*)
(* berechne den 1.1 des jahres von idate. *)
yr := year(idate);
d1 := year_begin(yr);
(* wochentag von d1 *)
w1 := weekday(d1);
(* offset des montags der eletzten KW des vorjahres *)
(* wenn der erste tag des jahres größer als donnerstag ist dann beginnt die letzte kw am montag davor *)
(* wenn der erste tag des jahres ein donnerstag oder kleiner ist beginnt die erste kw 2 montage davor *)
IF w1 < 5 THEN
	ds := DATE_TO_DWORD(d1) - (w1+6) * 86400;
ELSE
	ds := DATE_TO_DWORD(d1) + (1-w1) * 86400;
END_IF;

(* kalenderwoche des eingangsdatums *)
work_week := DWORD_TO_INT((DATE_TO_DWORD(idate) - ds) / 604800);

(* korrektur wenn work_week = 0 *)
IF work_week = 0 THEN
	(* work_week needs to be 53 when 1.jan of the year before is thursday or dec 31. is thursday. *)
	(* first and last weekday of a year is equal and one more day for a leap_year. *)
	IF w1 > 1 THEN w31 := w1 - 1; ELSE W31 := 7; END_IF;
	IF leap_year(yr - 1) THEN IF w31 > 1 THEN w01 := W31 - 1; ELSE w1 := 7; END_IF; END_IF;
	(* if first or last day of a year is a thursday, the year has 53 weeks *)
	IF w31 = 4 OR w01 = 4 THEN work_week := 53; ELSE work_week := 52; END_IF;
ELSE
	(* end of year calculation *)
	(* calculated the first and last weekday *)
	IF leap_year(yr) THEN
		IF w1 < 7 THEN w31 := w1 + 1; ELSE w31 := 1; END_IF;
	ELSE
		w31 := w1;
	END_IF;
	(* if first or last day is thursday then the year has 53 weeks otherwise only 52 *)
	IF w31 = 4 OR w1 = 4 THEN wm := 53; ELSE wm := 52; END_IF;
	IF work_week > wm THEN work_week := 1; END_IF;
END_IF;



(* old code before rev 1.2
w1 := weekday(set_Date(year(idate), 1,1));
IF w1 < 5 THEN
	work_week := (day_of_year(idate) + w1 + 5)/7;
ELSE
	work_week := (day_of_year(idate) + w1 - 2)/7;
END_IF
*)


(* revision history

hm 17.1.2007		rev 1.1
	deleted unused variable yday

hm	19. dec 2007	rev 1.2
	changed code for better performance
	changed code to comply with ISO8601
*)
END_FUNCTION

(* POU String/FIND_CHAR, ST *)
FUNCTION FIND_CHAR : INT
VAR_INPUT
	str : STRING;
	pos : INT;
END_VAR
VAR
	i: INT;
	pt : POINTER TO ARRAY[1..255] OF BYTE;
	stop: INT;
	X: BYTE;
END_VAR

(*
version 1.0	29. feb 2008
programmer 	hugo
tested by		tobias

find_char searches str and returns the starting position of the first character that is not a control character.
control characters are the ascii character 00 .. 31.

*)
pt := ADR(str);
stop := LEN(str);
FOR i := MAX(pos,1) TO stop DO;
	X := pt^[i];
	IF X > 31 THEN
		FIND_CHAR := i;
		RETURN;
	END_IF;
END_FOR;
FIND_CHAR := 0;


(* revision history
hm		29. feb 2008	rev 1.0
	original version

*)
END_FUNCTION

(* POU String/FIND_CTRL, ST *)
FUNCTION FIND_CTRL : INT
VAR_INPUT
	str : STRING;
	pos : INT;
END_VAR
VAR
	i: INT;
	pt : POINTER TO ARRAY[1..255] OF BYTE;
	stop: INT;
	x: BYTE;
END_VAR

(*
version 1.0	29. feb 2008
programmer 	hugo
tested by		tobias

find_ctrl searches str and returns the starting position of a control character
control characters are the ascii character 00 .. 31.

*)
pt := ADR(str);
stop := LEN(str);
FOR i := MAX(pos,1) TO stop DO;
	x := PT^[I];
	IF x < 32 THEN
		FIND_CTRL := i;
		RETURN;
	END_IF;
END_FOR;
FIND_CTRL := 0;


(* revision history
hm		29. feb 2008	rev 1.0
	original version

*)
END_FUNCTION

(* POU String/FINDP, ST *)
FUNCTION FINDP : INT
VAR_INPUT
	str : STRING;
	src : STRING;
	pos: INT;
END_VAR
VAR
	i: INT;
	ls: INT;
	lx: INT;
	stp: INT;
END_VAR

(*
version 1.1	29. feb 2009
programmer 	hugo
tested by		tobias

the function findP searches a string str for the occurence of src beginning at the position pos.

*)
ls := LEN(str);
lx := LEN(src);
IF ls < lx OR lx = 0 THEN RETURN; END_IF;
stp := ls - lx + 1;
FOR i := MAX(pos,1) TO stp DO
	IF MID(str,lx,i) = src THEN
		FINDP := i;
		RETURN;
	END_IF;
END_FOR;
FINDP := 0;

(* revision histroy
hm		4. feb. 2008	rev 1.0
	original release

hm		29. feb 2008	rev 1.1
	ADDED MAX(pos,1) in loop initialization

*)	
END_FUNCTION

(* POU XTEST/Ideas/FM_INVSQRT, ST *)
FUNCTION FM_INVSQRT : REAL
VAR_INPUT
	X: REAL;
END_VAR
VAR
	PTR : POINTER TO DWORD;
	XHALF: REAL;
END_VAR
XHALF := X * 0.5;
ptr := ADR(X);
ptr^ := 16#5F375A86 - SHR(ptr^,1);
FM_INVSQRT := X * (1.5 - XHALF * X * X);
END_FUNCTION

(* POU XTEST/Ideas/I2C, ST *)
FUNCTION_BLOCK I2C
VAR_INPUT
	scl_in : BOOL;
	sda_in : BOOL;
END_VAR
VAR_OUTPUT
	scl_out : BOOL;
	sda_out : BOOL;
	busy: BOOL;
	error: BOOL;
END_VAR
VAR
	state : INT;
END_VAR
(* the following state machine is responsible for all actions on the I2C Bus *)
CASE state OF
	0:	(* no actions *)
		busy := FALSE;

	1: (* ready for transfer *)
		RETURN;

	10: (* generate start condition *)
		busy := TRUE;
		IF sda_in AND scl_in THEN
			(* bus is free, start sequence can be completed *)
			sda_out := FALSE;
			state := 11;
		ELSIF NOT scl_in AND sda_in THEN
			(* if scl is low and sda is true then scl needs to go high first *)
			scl_out := TRUE;
		ELSIF NOT scl_in AND NOT sda_in THEN
			(* both scl and sda are low sda need to go high first *)
			sda_out := TRUE;
		ELSIF NOT scl_in AND NOT sda_in THEN
			(* both scl and sda are low scl need to go low first *)
			scl_out := FALSE;
		END_IF;
	11: (* second phase of start cycle, pull scl low *)
		scl_out := FALSE;
		state := 1;

	20:	(* generate stop condition *)
		busy := TRUE;
		IF scl_in AND NOT sda_in THEN
			(* scl is high and sda is low sequence can be completed *)
			sda_out := TRUE;
			state := 0;
		ELSIF NOT scl_in AND NOT sda_in THEN
			(* scl and sda are low,  scl need to go high first *)
			scl_out := TRUE;
		ELSIF NOT scl_in AND sda_in THEN
			(* scl is low and sda is high, sda need to go low first *)
			sda_out := FALSE;
		ELSIF scl_in AND sda_in THEN
			(* scl and sda are high, scl need to go low first *)
			scl_out := FALSE;
		END_IF;

	30:	(* master acknowledge cycle *)
		IF NOT busy AND scl_in THEN
			(* if no transfer takes place an acknowledge cannot be received *)
			error := TRUE;
		ELSIF TRUE THEN
			(* bring sda true to check for ack *)
			sda_out := TRUE;
		END_IF;



END_CASE
END_FUNCTION_BLOCK

(* POU Network/IP4_CHECK, ST *)
FUNCTION IP4_CHECK : BOOL
VAR_INPUT
	NIP : DWORD;
	LIP : DWORD;
	SM : DWORD;
END_VAR
VAR
END_VAR

(*
version 1.0	4. mar 2008
programmer 	hugo
tested by		oscat

IP4_CHECK testet ob eine Network IP und Local_IP im selben Subnet sind.

*)
IP4_CHECK := (NIP AND sm) = (LIP AND SM);


(* revision history
hm		4. mar 2008	rev 1.0
	original version

*)
END_FUNCTION

(* POU Network/IP4_DECODE, ST *)
FUNCTION IP4_DECODE : DWORD
VAR_INPUT
	str : STRING;
END_VAR
VAR
	d1, d2, d3, d4 : INT;
	s1, s2, s3, s4 : STRING(3);
END_VAR

(*
version 1.0	29. feb 2008
programmer 		kurt
tested by		hugo

IP4_DECODE testet ob ein string eine gültige IPv4 Adresse enthält und gibt die 4 Bytes der IP Adresse als DWORD zurück.

*)
IP4_DECODE := 0;
(* check wheather 3 dots are present *)
IF COUNT_CHAR(str,46) <> 3 THEN RETURN; END_IF;
(* store the positions of the 3 dots *)
d1 := FINDP(str,'.',1);
d2 := FINDP(str,'.',d1+1);
d3 := FINDP(str,'.',d2+1);
IF d1 > 4 OR d2 - d1 > 4 OR d3 - d2 > 4 THEN RETURN; END_IF;
(* store the 3 strings between the dots in d1 .. d4 *)
s1 := LEFT(str,d1-1);
s2 := MID(str,d2-d1-1,d1+1);
s3 := MID(str,d3-d2-1,d2+1);
s4 := RIGHT(str,LEN(str)-d3);
(* check if the 3 strings are numbers only *)
IF NOT IS_NUM(s1) OR NOT IS_NUM(s2) OR NOT IS_NUM(s3) OR NOT IS_NUM(s4) THEN RETURN; END_IF;
(* convert the 4 numbers and check range 0..255 *)
d1 := STRING_TO_INT(s1);
d2 := STRING_TO_INT(s2);
d3 := STRING_TO_INT(s3);
d4 := STRING_TO_INT(s4);
(* check range of numbers *)
IF d1 > 255 OR d2 > 255 OR d3 > 255 OR d4 > 255 THEN RETURN; END_IF;
(* convert to output *)
IP4_DECODE := SHL(INT_TO_DWORD(d1),24) OR SHL(INT_TO_DWORD(d2),16) OR SHL(INT_TO_DWORD(d3),8) OR INT_TO_DWORD(d4);



(* revision history
hm		29. feb 2008	rev 1.0
	original version

*)
END_FUNCTION

(* POU String/IS_NUM, ST *)
FUNCTION IS_NUM : BOOL
VAR_INPUT
	str : STRING;
END_VAR
VAR
	L : INT;
	pt : POINTER TO BYTE;
	pos: INT;
END_VAR

(*
version 1.0	29. feb 2008
programmer 		kurt
tested by		hugo

IS_NUM testet ob in einem string nur Zahlen 0..9 vorkommen.

*)
PT := ADR(str);
L := LEN(str);
FOR pos := 1 TO L DO
	IF NOT (ISC_NUM(pt^)) THEN
		IS_NUM := FALSE;
		RETURN;
	END_IF;
    	PT := PT + 1;
END_FOR;
IS_NUM := L > 0;


(* revision history
hm		29. feb 2008	rev 1.0
	original version

*)
END_FUNCTION

(* POU String/ISC_NUM, ST *)
FUNCTION ISC_NUM : BOOL
VAR_INPUT
	IN : BYTE;
END_VAR
VAR
END_VAR

(*
version 1.0	6. mar 2008
programmer 	oscat
tested by		hugo

ISC_NUM checks if a character is 0..9.

*)
ISC_NUM := IN > 47 AND IN < 58;

(* revision history
hm		6. mar. 2008	rev 1.0
	original version

*)
END_FUNCTION

(* POU Device Drivers/IRTRANS_1, ST *)
FUNCTION_BLOCK IRTRANS_1
VAR_INPUT CONSTANT
	device_code : STRING;
	key_code : STRING;
END_VAR
VAR_INPUT
	cmd : BOOL;
END_VAR
VAR_IN_OUT
	device : STRING;
	key : STRING;
END_VAR
VAR_OUTPUT
	Q : BOOL;
END_VAR
VAR
END_VAR

(*
	version 1.0	2 jan 2008
	programmer 	hugo
	tested BY		tobias

*)
IF cmd AND device_code = device AND key_code = key THEN
	Q := TRUE;
ELSE
	Q := FALSE;
END_IF;

(* revision history
hm	2. jan 2008		rev 1.0
	original version

*)
END_FUNCTION_BLOCK

(* POU Device Drivers/IRTRANS_4, ST *)
FUNCTION_BLOCK IRTRANS_4
VAR_INPUT CONSTANT
	device_code : STRING;
	key_code_0 : STRING;
	key_code_1 : STRING;
	key_code_2 : STRING;
	key_code_3 : STRING;
END_VAR
VAR_INPUT
	cmd : BOOL;
END_VAR
VAR_IN_OUT
	device : STRING;
	key : STRING;
END_VAR
VAR_OUTPUT
	Q0, Q1, Q2, Q3 : BOOL;
END_VAR
VAR
END_VAR

(*
	version 1.0	2 jan 2008
	programmer 	hugo
	tested BY		tobias

*)
Q0 := FALSE;
Q1 := FALSE;
Q2 := FALSE;
Q3 := FALSE;
IF cmd AND device_code = device THEN
	IF key = key_code_0 THEN q0 := TRUE;
	ELSIF key = key_code_1 THEN q1 := TRUE;
	ELSIF key = key_code_2 THEN q2 := TRUE;
	ELSIF key = key_code_3 THEN q3 := TRUE;
	END_IF;
END_IF;

(* revision history
hm	2. jan 2008		rev 1.0
	original version

*)
END_FUNCTION_BLOCK

(* POU Device Drivers/IRTRANS_8, ST *)
FUNCTION_BLOCK IRTRANS_8
VAR_INPUT CONSTANT
	device_code : STRING;
	key_code_0 : STRING;
	key_code_1 : STRING;
	key_code_2 : STRING;
	key_code_3 : STRING;
	key_code_4 : STRING;
	key_code_5 : STRING;
	key_code_6 : STRING;
	key_code_7 : STRING;
END_VAR
VAR_INPUT
	cmd : BOOL;
END_VAR
VAR_IN_OUT
	device : STRING;
	key : STRING;
END_VAR
VAR_OUTPUT
	Q0, Q1, Q2, Q3, Q4, Q5, Q6, Q7 : BOOL;
END_VAR
VAR
END_VAR

(*
	version 1.0	2 jan 2008
	programmer 	hugo
	tested BY		tobias

*)
Q0 := FALSE;
Q1 := FALSE;
Q2 := FALSE;
Q3 := FALSE;
Q4 := FALSE;
Q5 := FALSE;
Q6 := FALSE;
Q7 := FALSE;
IF cmd AND device_code = device THEN
	IF key = key_code_0 THEN q0 := TRUE;
	ELSIF key = key_code_1 THEN q1 := TRUE;
	ELSIF key = key_code_2 THEN q2 := TRUE;
	ELSIF key = key_code_3 THEN q3 := TRUE;
	ELSIF key = key_code_4 THEN q4 := TRUE;
	ELSIF key = key_code_5 THEN q5 := TRUE;
	ELSIF key = key_code_6 THEN q6 := TRUE;
	ELSIF key = key_code_7 THEN q7 := TRUE;
	END_IF;
END_IF;

(* revision history
hm	2. jan 2008		rev 1.0
	original version

*)
END_FUNCTION_BLOCK

(* POU Device Drivers/IRTRANS_DECODE, ST *)
FUNCTION_BLOCK IRTRANS_DECODE
VAR_INPUT
	buffer : POINTER TO ARRAY[0..32000] OF BYTE;
END_VAR
VAR_IN_OUT
	length : DINT;
END_VAR
VAR_OUTPUT
	cmd : BOOL;
	device : STRING;
	key : STRING;
	error : BOOL;
END_VAR
VAR
	pt : POINTER TO BYTE;
	i : INT;
	stop : INT;
END_VAR

(*
	version 1.0	2 jan 2008
	programmer 	hugo
	tested BY		tobias

*)
(* do nothing if the buffer is empty *)
IF length > 0 THEN
	i := 0;
	error := TRUE;
	stop := DINT_TO_INT(length) - 2;
	(* read characters before first comma and store in device *)
	pt := ADR(device);
	WHILE i < stop DO
		IF buffer^[i] = 44 THEN EXIT; END_IF;
		pt^ := buffer^[i];
		pt := pt + 1;
		i := i + 1;
	END_WHILE;
	(* terminate the device string *)
	pt^ := 0;
	(* read after first comma and store in key *)
	i := i + 1;
	pt := ADR(key);
	WHILE i < stop DO
		pt^ := buffer^[i];
		pt := pt + 1;
		i := i + 1;
	END_WHILE;
	(* terminate the key string *)
	pt^:= 0;
	(* check if last two characters are $R$N 13, 10 *)
	IF buffer^[i] <> 13 AND buffer^[i+1] <> 10 THEN	RETURN;	END_IF;
	(* check if device and key are present *)
	IF LEN(device) = 0 OR LEN(key) = 0 THEN RETURN; END_IF;
	(* a valid transmission has been received *)
	cmd := TRUE;
	error := FALSE;
	(* clear the input buffer to allow the next transmission to occur *)
	length := 0;
ELSE
	error := FALSE;
	cmd := FALSE;
END_IF;


(* revision history
hm	2. jan 2008		rev 1.0
	original version

*)
END_FUNCTION_BLOCK

(* POU String/IS_ALNUM, ST *)
FUNCTION IS_ALNUM : BOOL
VAR_INPUT
	str : STRING;
END_VAR
VAR
	L: INT;
	pt : POINTER TO BYTE;
	pos: INT;
END_VAR

(*
version 1.0	29. feb 2008
programmer 		kurt
tested by		hugo

ISC_ALNUM testet ob in einem string nur Zahlen 0..9 vorkommen.

*)
PT := ADR(str);
L := LEN(str);
FOR pos := 1 TO L DO
	IF NOT (ISC_ALPHA(pt^) OR ISC_NUM(pt^)) THEN
		IS_ALNUM := FALSE;
		RETURN;
	END_IF;
    	PT := PT + 1;
END_FOR;
IS_ALNUM := L > 0;


(* revision history
hm		29. feb 2008	rev 1.0
	original version

*)
END_FUNCTION

(* POU String/ISC_ALPHA, ST *)
FUNCTION ISC_ALPHA : BOOL
VAR_INPUT
	IN : BYTE;
END_VAR
VAR
END_VAR

(*
version 1.0	6. mar 2008
programmer 	oscat
tested by		hugo

ISC_ALPHA checks if a character is a..z or A..Z.

*)
IF extended_ascii THEN
	ISC_ALPHA := (in > 64 AND in < 91) OR (in > 191  AND in <> 215 AND in <> 247) OR (in > 96 AND in < 123);
ELSE
	ISC_ALPHA := (IN > 64 AND IN < 91) OR (in > 96 AND in < 123);
END_IF;

(* revision history
hm		6. mar. 2008	rev 1.0
	original version

*)
END_FUNCTION

(* POU String/IS_ALPHA, ST *)
FUNCTION IS_ALPHA : BOOL
VAR_INPUT
	str : STRING;
END_VAR
VAR
	L: INT;
	pt : POINTER TO BYTE;
	pos: INT;
END_VAR

(*
version 1.0	29. feb 2008
programmer 		kurt
tested by		hugo

IS_ALPHA testet ob in einem string nur Zeichen a-z oder A - Z vorkommen.

*)
PT := ADR(str);
L := LEN(str);
FOR pos := 1 TO L DO
	IF NOT ISC_ALPHA(pt^) THEN
		IS_ALPHA := FALSE;
		RETURN;
	END_IF;
    	PT := PT + 1;
END_FOR;
IS_ALPHA := L > 0;


(* revision history
hm		29. feb 2008	rev 1.0
	original version

*)
END_FUNCTION

(* POU String/IS_CTRL, ST *)
FUNCTION IS_CTRL : BOOL
VAR_INPUT
	str : STRING;
END_VAR
VAR
	L: INT;
	pt : POINTER TO BYTE;
	pos: INT;
END_VAR

(*
version 1.0	29. feb 2008
programmer 		kurt
tested by		hugo

IS_CTRL testet ob in einem string nur Steuerzeichen (Char < 32) vorkommen.

*)
PT := ADR(str);
L := LEN(str);
FOR pos := 1 TO L DO
	IF NOT (ISC_CTRL(pt^)) THEN
		IS_CTRL := FALSE;
		RETURN;
	END_IF;
    	PT := PT + 1;
END_FOR;
IS_CTRL := L > 0;


(* revision history
hm		29. feb 2008	rev 1.0
	original version

*)
END_FUNCTION

(* POU String/ISC_CTRL, ST *)
FUNCTION ISC_CTRL : BOOL
VAR_INPUT
	IN : BYTE;
END_VAR
VAR
END_VAR

(*
version 1.0	6. mar 2008
programmer 	oscat
tested by		hugo

ISC_ALPHA checks if a character is a control character.

*)
ISC_CTRL := IN < 32 OR IN = 127;

(* revision history
hm		6. mar. 2008	rev 1.0
	original version

*)
END_FUNCTION

(* POU String/IS_HEX, ST *)
FUNCTION IS_HEX : BOOL
VAR_INPUT
	str : STRING;
END_VAR
VAR
	L: INT;
	pt : POINTER TO BYTE;
	pos: INT;
END_VAR

(*
version 1.0	29. feb 2008
programmer 		kurt
tested by		hugo

IS_HEX testet ob in einem string nur Zahlen 0..9 oder A..F oder a..f  vorkommen.

*)
PT := ADR(str);
L := LEN(str);
FOR pos := 1 TO L DO
	IF NOT (ISC_HEX(pt^)) THEN
		IS_HEX := FALSE;
		RETURN;
	END_IF;
    	PT := PT + 1;
END_FOR;
IS_HEX := L > 0;


(* revision history
hm		29. feb 2008	rev 1.0
	original version

*)
END_FUNCTION

(* POU String/ISC_HEX, ST *)
FUNCTION ISC_HEX : BOOL
VAR_INPUT
	IN : BYTE;
END_VAR
VAR
END_VAR

(*
version 1.0	6. mar 2008
programmer 	oscat
tested by		hugo

ISC_HEX checks if a character is 0..9, A..F, a..f.

*)
ISC_HEX := (IN > 47 AND IN < 58) OR (IN > 64 AND IN < 71) OR (IN > 96 AND IN < 103);

(* revision history
hm		6. mar. 2008	rev 1.0
	original version

*)
END_FUNCTION

(* POU Network/IS_IP4, ST *)
FUNCTION IS_IP4 : BOOL
VAR_INPUT
	str : STRING;
END_VAR
VAR
END_VAR

(*
version 1.0	1. mar 2008
programmer 		kurt
tested by		hugo

IS_IP4 testet ob ein string eine gültige IPv4 Adresse enthält.

*)
IS_IP4 := IP4_DECODE(str) > 0;


(* revision history
hm		1. mar 2008	rev 1.0
	original version

*)
END_FUNCTION

(* POU String/IS_LOWER, ST *)
FUNCTION IS_LOWER : BOOL
VAR_INPUT
	str : STRING;
END_VAR
VAR
	l: INT;
	pt : POINTER TO BYTE;
	pos: INT;
END_VAR

(*
version 1.0	29. feb 2008
programmer 		kurt
tested by		hugo

IS_LOWER testet ob in einem string nur kleinbuchstaben vorkommen.

*)
PT := ADR(str);
L := LEN(str);
FOR pos := 1 TO L DO
	IF NOT (ISC_LOWER(pt^)) THEN
		IS_LOWER := FALSE;
		RETURN;
	END_IF;
    	PT := PT + 1;
END_FOR;
IS_LOWER := L > 0;


(* revision history
hm		29. feb 2008	rev 1.0
	original version

*)
END_FUNCTION

(* POU String/ISC_LOWER, ST *)
FUNCTION ISC_LOWER : BOOL
VAR_INPUT
	IN : BYTE;
END_VAR
VAR
END_VAR

(*
version 1.0	6 mar 2008
programmer 	hugo
tested by		tobias

isc_lower checks if a character is lowercase.

*)
IF extended_ascii THEN
	ISC_LOWER := ((in > 96) AND (in < 123)) OR ((in > 222) AND (in <> 247));
ELSE
	ISC_LOWER := ((in > 96) AND (in < 123));
END_IF;

(* revision history
hm		6. mar 2008	rev 1.0
	original version

*)
END_FUNCTION

(* POU String/IS_UPPER, ST *)
FUNCTION IS_UPPER : BOOL
VAR_INPUT
	str : STRING;
END_VAR
VAR
	L: INT;
	pt : POINTER TO BYTE;
	pos: INT;
END_VAR

(*
version 1.0	29. feb 2008
programmer 		kurt
tested by		hugo

IS_UPPER testet ob in einem string keine Kleinbuchstaben vorkommen.

*)
PT := ADR(str);
L := LEN(str);
FOR pos := 1 TO L DO
	IF NOT (ISC_UPPER(pt^)) THEN
		IS_UPPER := FALSE;
		RETURN;
	END_IF;
    	PT := PT + 1;
END_FOR;
IS_UPPER := L > 0;


(* revision history
hm		29. feb 2008	rev 1.0
	original version

*)
END_FUNCTION

(* POU String/ISC_UPPER, ST *)
FUNCTION ISC_UPPER : BOOL
VAR_INPUT
	IN : BYTE;
END_VAR
VAR
END_VAR

(*
version 1.0	6 mar 2008
programmer 	hugo
tested by		tobias

ISC_upper checks if a character is uppercase

*)
IF extended_ascii THEN
	ISC_UPPER :=  ((in > 64) AND (in < 91)) OR (((in > 191) AND (in < 223)) AND (in <> 215));
ELSE
	ISC_UPPER := ((in > 64) AND (in < 91));
END_IF;


(* revision history
hm		6. mar 2008	rev 1.0
	original version

*)
END_FUNCTION

(* POU XTEST/Performance Test/measure_times, ST *)
FUNCTION_BLOCK measure_times
VAR_INPUT
END_VAR
VAR_OUTPUT
END_VAR
VAR
	times, mn, mx : ARRAY[0..300] OF REAL;
	tx: DWORD;
	init: BOOL;
	last: DWORD;
	t_max: DWORD := 100;
	cycles: DWORD;
	c_max: DWORD := 10000;
	i: INT;
	stop: INT := 3;
	overhead: REAL;
	runx : fc_list;
	timex: REAL;
END_VAR
IF NOT init THEN
	init := TRUE;
	_array_init(ADR(mn),SIZEOF(mn),99999);
END_IF;

IF i > stop THEN i := 0; END_IF;
(* measure overhead *)
last := TIME_TO_DWORD(TIME());
tx := 0;
cycles := 0;
WHILE tx < t_max AND cycles < c_max DO
	runx(num := i, check := TRUE);
	tx := TIME_TO_DWORD(TIME()) - last;
	cycles := cycles + 1;
END_WHILE;
overhead := DWORD_TO_REAL(tx) * 1000.0 / cycles;

(* measure execution time *)
last := TIME_TO_DWORD(TIME());
tx := 0;
cycles := 0;
WHILE tx < t_max AND cycles < c_max DO
	runx(num := i, check := FALSE);
	tx := TIME_TO_DWORD(TIME()) - last;
	cycles := cycles + 1;
END_WHILE;
timex := DWORD_TO_REAL(tx) * 1000.0 / cycles - overhead;

(* berechne korrekturwert für if anweisung für ckeck *)
IF i = 0 THEN
	mn[0] := MIN(timex,mn[0]);
	mx[0] := MAX(timex,mx[0]);
	times[0] := round((mx[0] + mn[0])/2,2);
ELSE
	mn[i] := MIN(timex - times[0], mn[i]);
	mx[i] := MAX(timex - times[0], mx[i]);
	times[i] := round((mx[i] + mn[i])/2,1);
END_IF;

i := i + 1;
END_FUNCTION_BLOCK

(* POU String/MIRROR, ST *)
FUNCTION MIRROR : STRING
VAR_INPUT
	str : STRING;
END_VAR
VAR
	pi : POINTER TO ARRAY[1..255] OF BYTE;
	po : POINTER TO BYTE;
	lx: INT;
	i: INT;
END_VAR

(*
version 1.0	4 feb 2008
programmer 	hugo
tested by		tobias

this function reverses an input string.

*)
pi := ADR(str);
po := ADR(mirror);
lx := LEN(str);
FOR i := lx TO 1 BY - 1 DO
	po^ := pi^[i];
	po := po + 1;
END_FOR;
(* close output string *)
po^:= 0;


(* revision histroy
hm		4. feb. 2008		rev 1.0
	original release

*)	
END_FUNCTION

(* POU XTEST/Testprojekt/network_test, ST *)
FUNCTION_BLOCK network_test
VAR_INPUT
END_VAR
VAR_OUTPUT
	good : BOOL;
END_VAR
VAR CONSTANT
END_VAR
VAR
END_VAR
good := TRUE;

(* test ip4_decode *)
good := good AND IP4_DECODE('0.0.0.0') = 0;
good := good AND IP4_DECODE('1.2.3.4') = 16#01_02_03_04;
good := good AND IP4_DECODE('255.255.255.255') = 16#FF_FF_FF_FF;
good := good AND IP4_DECODE('256.188.3.4') = 0;
good := good AND IP4_DECODE('1.256.3.4') = 0;
good := good AND IP4_DECODE('1.2.256.4') = 0;
good := good AND IP4_DECODE('1.2.3.256') = 0;
good := good AND IP4_DECODE('1.2.3.4.') = 0;
good := good AND IP4_DECODE('.1.2.3.4.') = 0;
good := good AND IP4_DECODE('1.2.3') = 0;
good := good AND IP4_DECODE('1.A.3.4.') = 0;

(* test is_ip4 *)
good := good AND IS_IP4('0.0.0.0') = FALSE;
good := good AND IS_IP4('192.2.3.0') = TRUE;
good := good AND IS_IP4('255.255.255.255') = TRUE;
good := good AND IS_IP4('256.188.3.4') = FALSE;
good := good AND IS_IP4('1.256.3') = FALSE;
good := good AND IS_IP4('1.A.256.4') = FALSE;
good := good AND IS_IP4('251.188.3.4.1') = FALSE;

(* test ip4_check *)
good := good AND IP4_CHECK(16#01010101,16#01010102,16#FFFFFF00) = TRUE;
good := good AND IP4_CHECK(16#02010101,16#01010102,16#FFFFFF00) = FALSE;
good := good AND IP4_CHECK(16#01020101,16#01010102,16#FF000000) = TRUE;
good := good AND IP4_CHECK(16#02020202,16#01010101,16#000000) = TRUE;
END_FUNCTION_BLOCK

(* POU Other/Oscat_version, ST *)
FUNCTION Oscat_version : DWORD
VAR_INPUT
	in : BOOL;
END_VAR
VAR
END_VAR


(*
version 1.1	16 dec 2007
programmer 	hugo
tested by		tobias

oscat_version returns the version number in dword format
132 is library version 1.32
if IN = true, the release date will be returned

*)
IF in THEN
	Oscat_version := DATE_TO_DWORD(D#2008-3-15);
ELSE
	Oscat_version := 272;
END_IF;

(* revision history
hm	6. oct 2006	rev 1.0
	original version

hm	16. dec 2007	rev 1.1
	added possibility to return date and version depending on IN.
 
*)
END_FUNCTION

(* POU Engineering/signal processing/Range_to_Byte, ST *)
FUNCTION Range_to_Byte : BYTE
VAR_INPUT
	X : REAL;
	low : REAL;
	high : REAL;
END_VAR
VAR
END_VAR

(*
version 1.0	9. jan 2008
programmer 	hugo
tested by		tobias

Range_to_byte converts a real value between low and high into a byte

*)
Range_to_Byte := INT_TO_BYTE(TRUNC((LIMIT(low,X,high)-low) * 255.0 / (high - low)));


(* revision history
hm	9. jan 2008		rev 1.0
	original version

*)
END_FUNCTION

(* POU Engineering/signal processing/Range_to_Word, ST *)
FUNCTION Range_to_Word : WORD
VAR_INPUT
	X : REAL;
	low : REAL;
	high : REAL;
END_VAR
VAR
END_VAR

(*
version 1.0	9. jan 2008
programmer 	hugo
tested by		tobias

Range_to_word converts a real value between low and high into a byte

*)
Range_to_Word := DINT_TO_WORD(TRUNC((LIMIT(low,X,high)-low) * 65535.0 / (high - low)));


(* revision history
hm	9. jan 2008		rev 1.0
	original version

*)
END_FUNCTION

(* POU XTEST/Baustein Tests/rdm_test, ST *)
FUNCTION_BLOCK rdm_test
VAR_INPUT
END_VAR
VAR_OUTPUT
END_VAR
VAR
	x: REAL;
	mx: REAL;
	Mn: REAL;
	x0, x1,x2, x3, x4, x5,x6, x7,x8, x9: REAL;
	V, U : REAL;
	W, G : REAL;
	C: DINT;
	CX0, cx1, cx2, cx3, cx4, cx5, cx6,cx7,cx8,cx9: REAL;
	CV: REAL;
	CU: REAL;
	CW : REAL;
	CG : REAL;
	last : ARRAY[0..11] OF REAL;
	sum : ARRAY[0..11] OF REAL;
	start: ARRAY[1..50] OF REAL;
	index: INT;
	sum1, sum2, sum3, sum4, sum5,sum6,sum7,sum8,sum9: REAL;
	last1, last2, last3, last4, last5, last6, last7, last8, last9: REAL;
	delta: REAL;
	d0, d1, d2, d3, d4, d5, d6,d7,d8,d9: REAL;
	dX0, dx1, dx2, dx3, dx4, dx5, dx6, dx7, dx8, dx9: REAL;
	d20, d21, d22, d23, d24, d25, d26,d27,d28,d29: REAL;
	dX20, dx21, dx22, dx23, dx24, dx25, dx26, dx27, dx28, dx29: REAL;
	oldtime: DWORD;
END_VAR
IF T_PLC_MS() = oldtime THEN RETURN; END_IF;
oldtime := T_PLC_MS();

C := c + 1;
x := RDM(x);
(* check if X is less then 0 or 1 or higher which is not allowed *)
IF X < 0 THEN Mn := mn +1;
ELSIF X >= 1 THEN mx := mx +1;

(* check distribution*)
ELSIF X < 0.1 THEN	x0 := x0+1; CX0 := C/10/x0;
ELSIF X < 0.2 THEN	x1 := x1+1; CX1 := C/10/x1;
ELSIF X < 0.3 THEN	x2 := x2+1; CX2 := C/10/x2;
ELSIF X < 0.4 THEN	x3 := x3+1; CX3 := C/10/x3;
ELSIF X < 0.5 THEN	x4 := x4+1; CX4 := C/10/x4;
ELSIF X < 0.6 THEN	x5 := x5+1; CX5 := C/10/x5;
ELSIF X < 0.7 THEN	x6 := x6+1; CX6 := C/10/x6;
ELSIF X < 0.8 THEN	x7 := x7+1; CX7 := C/10/x7;
ELSIF X < 0.9 THEN	x8 := x8+1; CX8 := C/10/x8;
ELSIF X < 1 THEN		x9 := x9+1; CX9 := C/10/x9;
END_IF;


(* check near 0 *)
IF X < 0.01 THEN V := V +1; END_IF; CV := C/100/V;
IF X < 0.001 THEN U := U +1; END_IF; CU := C/1000/U;

(* check near 1 *)
IF X >= 0.99 THEN W := W + 1; END_IF;CW := C/100/V;
IF X >= 0.999 THEN G := G + 1; END_IF; CG := C/1000/G;

(* check sequence1 *)
index := DINT_TO_INT(C MOD 12);
sum[index] := sum[index] + last[index] - X;
last[index] := X;

(* check sequence2 and delta to be distributed evenly *)
delta := last1 - X;
sum1 := sum1 + delta;
IF ABS(delta) < 0.1 THEN	d0 := d0+1; dX0 := C/10/d0;
ELSIF ABS(delta) < 0.2 THEN	d1 := d1+1; dX1 := C/10/d1;
ELSIF ABS(delta) < 0.3 THEN	d2 := d2+1; dX2 := C/10/d2;
ELSIF ABS(delta) < 0.4 THEN	d3 := d3+1; dX3 := C/10/d3;
ELSIF ABS(delta) < 0.5 THEN	d4 := d4+1; dX4 := C/10/d4;
ELSIF ABS(delta) < 0.6 THEN	d5 := d5+1; dX5 := C/10/d5;
ELSIF ABS(delta) < 0.7 THEN	d6 := d6+1; dX6 := C/10/d6;
ELSIF ABS(delta) < 0.8 THEN	d7 := d7+1; dX7 := C/10/d7;
ELSIF ABS(delta) < 0.9 THEN	d8 := d8+1; dX8 := C/10/d8;
ELSIF ABS(delta) < 1 THEN   d9 := d9+1; dX9 := C/10/d9;
END_IF;
last1 := X;


IF c MOD 2 = 0 THEN
	delta := last2 - X;
	sum2 := sum2 + delta;
	IF ABS(delta) < 0.1 THEN	d20 := d20+1; dX20 := C/20/d20;
	ELSIF ABS(delta) < 0.2 THEN	d21 := d21+1; dX21 := C/20/d21;
	ELSIF ABS(delta) < 0.3 THEN	d22 := d22+1; dX22 := C/20/d22;
	ELSIF ABS(delta) < 0.4 THEN	d23 := d23+1; dX23 := C/20/d23;
	ELSIF ABS(delta) < 0.5 THEN	d24 := d24+1; dX24 := C/20/d24;
	ELSIF ABS(delta) < 0.6 THEN	d25 := d25+1; dX25 := C/20/d25;
	ELSIF ABS(delta) < 0.7 THEN	d26 := d26+1; dX26 := C/20/d26;
	ELSIF ABS(delta) < 0.8 THEN	d27 := d27+1; dX27 := C/20/d27;
	ELSIF ABS(delta) < 0.9 THEN	d28 := d28+1; dX28 := C/20/d28;
	ELSIF ABS(delta) < 1 THEN   d29 := d29+1; dX29 := C/20/d29;
	END_IF;
	last2 := X;
END_IF;
IF c MOD 3 = 0 THEN
	sum3 := sum3 + last3 - x; last3 := X;
END_IF;
IF c MOD 4 = 0 THEN
	sum4 := sum4 + last4 - x; last4 := X;
END_IF;
IF c MOD 5 = 0 THEN
	sum5 := sum5 + last5 - x; last5 := X;
END_IF;
IF c MOD 6 = 0 THEN
	sum6 := sum6 + last6 - x; last6 := X;
END_IF;
IF c MOD 7 = 0 THEN
	sum7 := sum7 + last7 - x; last7 := X;
END_IF;
IF c MOD 8 = 0 THEN
	sum8 := sum8 + last8 - x; last8 := X;
END_IF;
IF c MOD 9 = 0 THEN
	sum9 := sum9 + last9 - x; last9 := X;
END_IF;

(* store startup sequence *)
IF c <= 50 THEN
	start[DINT_TO_INT(C)] := X;
END_IF;
END_FUNCTION_BLOCK

(* POU String/REPLACE_ALL, ST *)
FUNCTION REPLACE_ALL : STRING
VAR_INPUT
	str : STRING;
	src : STRING;
	rep : STRING;
END_VAR
VAR
	pos: INT;
	lp : INT;
	lx : INT;
END_VAR

(*
version 1.0	4 feb 2008
programmer 	hugo
tested by		tobias

the function findP searches a string str for the occurence of src beginning at the position pos.

*)
REPLACE_ALL := str;
lx := LEN(src);
lp := LEN(rep);
pos := FINDP(REPLACE_ALL, src, 1);
WHILE pos > 0 DO
	REPLACE_ALL := REPLACE(REPLACE_ALL,rep,lx, pos);
	pos := FINDP(REPLACE_ALL, src, pos + lp);
END_WHILE;

(* revision histroy
hm		4. feb. 2008		rev 1.0
	original release

*)	
END_FUNCTION

(* POU String/REPLACE_UML, ST *)
FUNCTION REPLACE_UML : STRING
VAR_INPUT
	str : STRING;
END_VAR
VAR
	l : INT;
	pt : POINTER TO BYTE;
	pto : POINTER TO BYTE;
	pos : INT;
END_VAR

(*
version 1.0	29. feb 2008
programmer 		kurt
tested by		hugo

REPLACE_UML replaces all occurences of Ä,Ö,Ü and ä,ö,ü,ß with Ae, ae, Oe, oe, Ue, ue and ss.

*)
PT := ADR(str);
pto := ADR(REPLACE_UML);
l := LEN(str);
FOR pos := 1 TO l DO
	IF PT^ = 196 OR PT^ = 214 OR PT^ = 220 OR PT^ = 223 OR PT^ = 228 OR PT^ = 246 OR PT^ = 252 THEN
		IF pt^ > 223 THEN
			IF pt^ = 228 THEN
				pto^ := 97;
				pto := pto + 1;
				pto^ := 101;
				pto := pto + 1;
			ELSIF pt^ = 246 THEN
				pto^ := 111;
				pto := pto + 1;
				pto^ := 101;
				pto := pto + 1;
			ELSE
				pto^ := 117;
				pto := pto + 1;
				pto^ := 101;
				pto := pto + 1;
			END_IF;
		ELSE
			IF pt^ = 196 THEN
				pto^ := 65;
				pto := pto + 1;
				pto^ := 101;
				pto := pto + 1;
			ELSIF pt^ = 214 THEN
				pto^ := 79;
				pto := pto + 1;
				pto^ := 101;
				pto := pto + 1;
			ELSIF pt^ = 220 THEN
				pto^ := 85;
				pto := pto + 1;
				pto^ := 101;
				pto := pto + 1;
			ELSIF pt^ = 223 THEN
				pto^ := 115;
				pto := pto + 1;
				pto^ := 115;
				pto := pto + 1;
			END_IF;
		END_IF;
	ELSE
		pto^ := pt^;
		pto := pto + 1;
	END_IF;
PT := PT + 1;
END_FOR;
(* properly close the output string *)
pto^ := 0;


(* revision history
hm		29. feb 2008	rev 1.0
	original version

*)
END_FUNCTION

(* POU Time&Date/RTC_2, ST *)
FUNCTION_BLOCK RTC_2
VAR_INPUT
	SET : BOOL;
	SDT : DT;
	SMS : INT;
	DEN : BOOL;
	OFS : INT;
END_VAR
VAR_OUTPUT
	UDT : DT;
	LDT : DT;
	DSO : BOOL;
	XMS : INT;
END_VAR
VAR
	RT : RTC_MS;
	T: INT;
END_VAR

(*
version 1.1	20. feb. 2008
programmer 	hugo
tested by	tobias

RTC_2 is a real time clock module which runs utc and generates local time from utc.
daylight savings time can be enabled with den and an additional local time is generated with a delay of ofs.

*)
(* call rtc *)
RT(SET := SET, SDT := SDT, SMS := SMS);
UDT := rt.xdt;
XMS := rt.XMS;

(* check for daylight savings time and set dso output *)
dso := DST(udt) AND DEN;
IF dso THEN T := 1; ELSE T := 0; END_IF;

(* calculate time offset and set ldt output *)
LDT := DWORD_TO_DT(DT_TO_DWORD(UDT) + INT_TO_DWORD(ofs + T) * 3600);


(* revision history
hm		20. jan. 2008	rev 1.0
	original version

hm		20. feb. 2008	rev 1.1
	added Millisecond Set input
*)
END_FUNCTION_BLOCK

(* POU Time&Date/RTC_MS, ST *)
FUNCTION_BLOCK RTC_MS
VAR_INPUT
	SET : BOOL;
	SDT : DT;
	SMS : INT;
END_VAR
VAR_OUTPUT
	XDT : DT;
	XMS : INT;
END_VAR
VAR
	init: BOOL;
	last: DWORD;
	Tx: DWORD;
END_VAR

(*
version 1.1	20. feb. 2008
programmer 	hugo
tested by	tobias

RTC_MS is a real time clock module which can be set to SDT when set is TRUE and the outputs XDT and XT present the DateTime and TOD with a resolution of milliseconds.

*)
tx := T_PLC_MS();
IF set OR NOT init THEN
	(* clock needs to be set when set is true or after power up *)
	init := TRUE;
	xdt := SDT;
	XMS := SMS;
ELSE
	XMS := XMS + DWORD_TO_INT(tx - last);
	(* check if one second has expired *)
	IF XMS > 999 THEN
		XDT := XDT + T#1s;
		XMS := XMS - 1000;
	END_IF;
END_IF;
last := tx;


(* revision history
hm		20. jan. 2008	rev 1.0
	original version

hm		20. feb. 2008	rev 1.1
	added Millisecond Set input
*)
END_FUNCTION_BLOCK

(* POU Logic/FF edge triggered/select_8, ST *)
FUNCTION_BLOCK select_8
VAR_INPUT
	EN : BOOL;
	SET : BOOL;
	IN : BYTE;
	UP : BOOL;
	DN : BOOL;
	RST : BOOL;
END_VAR
VAR_OUTPUT
	Q0, Q1, Q2, Q3, Q4, Q5, Q6, Q7 : BOOL;
		STATE : INT;
END_VAR
VAR
	last_up: BOOL;
	last_dn : BOOL;
END_VAR

(*
	version 1.0	16 jan 2008
	programmer 	hugo
	tested BY	tobias

select_8 selects one of 8 outputs at any time. the outputscan be selected by up or down keys and an independent anable switches all outouts off if set false


*)
IF rst THEN
	state := 0;
ELSIF set THEN
	state := IN;
ELSIF up AND NOT last_up THEN
	state := inc(state,1,7);
ELSIF dn AND NOT last_dn THEN
	state := inc(state,-1,7);
END_IF;
last_UP := UP;
last_DN := DN;

Q0 := FALSE;
Q1 := FALSE;
Q2 := FALSE;
Q3 := FALSE;
Q4 := FALSE;
Q5 := FALSE;
Q6 := FALSE;
Q7 := FALSE;

IF en THEN
	CASE state OF
		0: Q0 := TRUE;
		1: Q1 := TRUE;
		2: Q2 := TRUE;
		3: Q3 := TRUE;
		4: Q4 := TRUE;
		5: Q5 := TRUE;
		6: Q6 := TRUE;
		7: Q7 := TRUE;
	END_CASE;
END_IF;

(* revision history
hm	16. jan 2008	rev 1.0
	original version

*)
END_FUNCTION_BLOCK

(* POU XTEST/Baustein Tests/set_date_test, ST *)
FUNCTION_BLOCK set_date_test
VAR_INPUT
END_VAR
VAR_OUTPUT
	OK : BOOL;
	rx : DWORD;
	fdate : DATE;
END_VAR
VAR
	yr : INT;
	last: REAL;
	day: INT;
	i: INT;
	temp: DATE;
	init: BOOL;
	mth: INT;
END_VAR
IF NOT init THEN
	ok := TRUE;
	init := TRUE;
END_IF;
FOR i := 1 TO 1000 DO
	last := RDM(last);
	yr := TRUNC(last * 130 + 1970);
	last := RDM(last);
	mth := TRUNC(last * 11.999) + 1;
	last := RDM(last);
	day := TRUNC(last * 30.999) + 1;
	CASE mth OF
		2 : IF leap_year(yr) THEN IF day > 29 THEN day := 29; END_IF;	ELSE IF day > 28 THEN day := 28; END_IF; END_IF;
		4 : IF day > 30 THEN day := 30; END_IF;
		6 : IF day > 30 THEN day := 30; END_IF;
		9 : IF day > 30 THEN day := 30; END_IF;
		11 : IF day > 30 THEN day := 30; END_IF;
	END_CASE;
	temp := set_Date(yr,mth,day);
	IF month(temp) <> mth THEN
		ok := FALSE;
		fdate := temp;
	END_IF;
	IF year(temp) <> yr THEN
		ok := FALSE;
		fdate := temp;
	END_IF;
	IF day_of_month(temp) <> day THEN
		ok := FALSE;
		fdate := temp;
	END_IF;
	rx := rx + 1;
END_FOR;
END_FUNCTION_BLOCK

(* POU XTEST/Ideas/sntp, ST *)
FUNCTION_BLOCK sntp
VAR_INPUT
	SET : BOOL;
END_VAR
VAR_OUTPUT
	TP :	BOOL;
	UDT :	UDINT;
	XMS :	INT;
	error :	BOOL;
END_VAR
(*
VAR_IN_OUT
	xStartSend :	BOOL;
	snd_length :	DINT;
	snd_buffer :	oscat_us_IP_DATA;
	rec_length :	DINT;
	rev_buffer :	oscat_us_IP_DATA;
END_VAR
VAR
	i :	INT;
	state :	INT;
	last :	UDINT;
	tx :	UDINT;
END_VAR *)
RETURN;
(*
(* read system time *)
tx := T_PLC_MS();

CASE state OF

00: (* Domain Name System (query) *)
  IF SET = FALSE THEN RETURN; END_IF;

  snd_buffer.bya_IP_DATA[01] := BYTE#16#1B;
  FOR i := 2 TO 48 DO
    snd_buffer.bya_IP_DATA[i] := BYTE#16#00;
  END_FOR;

  snd_length := DINT#48;
  xStartSend := TRUE;  
  state := 01;
  TP := FALSE;
  error := FALSE;
  last := tx;

01:
  (* Receive Data - Timeout 6 sek. *)
  IF (tx - last) > UDINT#6000 THEN
    snd_length := DINT#00;
    state := 3;
    error := TRUE; (* Timeout *)
  END_IF;
  
  (* länge der empfangenen Daten prüfen *)
  IF rec_length  < DINT#48 THEN RETURN; END_IF;

  (* Umrechnung SNTP Timestamp Base 1900-01-01 mit Internet Byte-Order -> Unix 1970-01-01 = +2208988800 sekunden*)
  UDT := DWORD_TO_UDINT(DWord_of_Byte(rev_buffer.bya_IP_DATA[44],rev_buffer.bya_IP_DATA[43],rev_buffer.bya_IP_DATA[42],rev_buffer.bya_IP_DATA[41]))- UDINT#2208988800;

  (* Original-Sekundenanteile sind als 32 Bit Fractal dargestellt *) 
  (* ms nur mit veringerte Auflösung berechnen 1/65535 -> Highword verwenden *)

  (* schnelle Version: durch 64 dividieren -> führt zu ca 25ms Rechenfehler *)
  XMS := WORD_TO_INT(SHR_WORD(Word_of_Byte(rev_buffer.bya_IP_DATA[46],rev_buffer.bya_IP_DATA[45]),6));

  (* genauere Variante noch besser wäre / REAL#65.535 aber ......... 
  XMS := UINT_TO_INT(WORD_TO_UINT(Word_of_Byte(rev_buffer.bya_IP_DATA[46],rev_buffer.bya_IP_DATA[45])) / UINT#66);
  *)

  (* Zeitdifferenz (Laufzeitfehler) zwischen Send und Receive /2 teilen *)
  XMS := XMS + DWORD_TO_INT(SHR_DWORD(UDINT_TO_DWORD(tx - last),1));

  (* sekundenanteile der Zeitdifferenz *)
  UDT := UDT + INT_TO_UDINT(XMS / 1000);
  (* ms übernehmen *)
  XMS := XMS MOD 1000;

  snd_length := DINT#00;
  state := 2;
  TP := TRUE;

02:
  TP := FALSE;
  
  IF SET = FALSE THEN 
    state := 0;
    error := FALSE;
  END_IF;
END_CASE;

(*               SNTP Datenstruktur
                                  1                   2                   3
              0 1 2 3 4 5 6 7 8 9 0 1 2 3 4 5 6 7 8 9 0 1 2 3 4 5 6 7 8 9 0 1
             +-+-+-+-+-+-+-+-+-+-+-+-+-+-+-+-+-+-+-+-+-+-+-+-+-+-+-+-+-+-+-+-+
Byte: 01-04  |LI | VN  |Mode |    Stratum    |     Poll      |   Precision   |
             +-+-+-+-+-+-+-+-+-+-+-+-+-+-+-+-+-+-+-+-+-+-+-+-+-+-+-+-+-+-+-+-+
Byte: 05-08  |                          Root  Delay (32 Bit)                 |
             +-+-+-+-+-+-+-+-+-+-+-+-+-+-+-+-+-+-+-+-+-+-+-+-+-+-+-+-+-+-+-+-+
Byte: 09-12  |                       Root  Dispersion (32 Bit)               |
             +-+-+-+-+-+-+-+-+-+-+-+-+-+-+-+-+-+-+-+-+-+-+-+-+-+-+-+-+-+-+-+-+
Byte: 13-16  |                     Reference Identifier (32 Bit)             |
             +-+-+-+-+-+-+-+-+-+-+-+-+-+-+-+-+-+-+-+-+-+-+-+-+-+-+-+-+-+-+-+-+
Byte: 17-24  |                    Reference Timestamp (64 Bit)               |
             +-+-+-+-+-+-+-+-+-+-+-+-+-+-+-+-+-+-+-+-+-+-+-+-+-+-+-+-+-+-+-+-+
Byte: 25-32  |                    Originate Timestamp (64 Bit)               |
             +-+-+-+-+-+-+-+-+-+-+-+-+-+-+-+-+-+-+-+-+-+-+-+-+-+-+-+-+-+-+-+-+
Byte: 33-40  |                     Receive Timestamp (64 Bit)                |
             +-+-+-+-+-+-+-+-+-+-+-+-+-+-+-+-+-+-+-+-+-+-+-+-+-+-+-+-+-+-+-+-+
Byte: 41-48  |                     Transmit Timestamp (64 Bit)               |
             +-+-+-+-+-+-+-+-+-+-+-+-+-+-+-+-+-+-+-+-+-+-+-+-+-+-+-+-+-+-+-+-+
Byte: 49-52  |                 Key Identifier (optional) (32 Bit)            |
             +-+-+-+-+-+-+-+-+-+-+-+-+-+-+-+-+-+-+-+-+-+-+-+-+-+-+-+-+-+-+-+-+
Byte: 53-68  |                 Message Digest (optional) (128 Bit)           |
             +-+-+-+-+-+-+-+-+-+-+-+-+-+-+-+-+-+-+-+-+-+-+-+-+-+-+-+-+-+-+-+-+

*)

(*
Worldwide NTP-Server


NIST-Zeitserver
• time-a.nist.gov
129.6.15.28 
NIST, Gaithersburg, Maryland 
• time-a.nist.gov
129.6.15.28 
NIST, Gaithersburg, Maryland 
• time-a.timefreq.bldrdoc.gov
132.163.4.101 (Stand: 1. Dezember 1999)
NIST, Boulder, Colorado 
• time-b.timefreq.bldrdoc.gov
132.163.4.102 (Stand: 1. Dezember 1999)
NIST, Boulder, Colorado 
• time-c.timefreq.bldrdoc.gov
132.163.4.103 (Stand: 1. Dezember 1999)
NIST, Boulder, Colorado 
• utcnist.colorado.edu
128.138.140.44
University of Colorado, Boulder 
• time.nist.gov
192.43.244.18
NCAR, Boulder, Colorado 
• time-nw.nist.gov
131.107.1.10
Microsoft, Redmond, Washington 
• nist1.dc.certifiedtime.com
216.200.93.8
Abovnet, North Virginia 
• nist1.datum.com
209.0.72.7
Datum, San Jose, Kalifornien 
• nist1.nyc.certifiedtime.com
208.184.49.129 
Abovnet, New York City 
• nist1.sjc.certifiedtime.com
207.126.103.202
Abovnet, San Jose, Kalifornien 

Zeitserver der ersten Ebene
Sortiert nach Standort: 
Nordamerika
• Palo Alto, Kalifornien: Systems Research Center, Compaq Computer Corp.
204.123.2.72: usno.pa-x.dec.com; CNAME: navobs1.pa-x.dec.com
Servicebereich: US-Zeitzonen PST (Pacific Standard Time) und MST (Mountain Standard Time) 
• Marina del Rey, Kalifornien: USC Information Sciences Institute
128.9.176.30: timekeeper.isi.edu
Servicebereich: CalRen2- und Los Nettos-Bereich  
• Washington, DC: U.S. Naval Observatory
192.5.41.41: tock.usno.navy.mil 
192.5.41.40: tick.usno.navy.mil
Servicebereich: NSFNET 
• Ottawa, Ontario, Kanada: National Research Council of Canada
time.chu.nrc.ca
Servicebereich: Kanada 
• Raleigh, North Carolina: North Carolina State University
152.1.58.124: terrapin.csc.ncsu.edu
Servicebereich: Südosten der USA 
• Cambridge, Massachusetts: MIT Information Systems
18.72.0.3: bitsy.mit.edu 
Servicebereich: NSFNET- und NEARnet-Bereich 
• Cambridge, Massachusetts: MIT
18.26.4.105: bonehed.lcs.mit.edu
Servicebereich: Osten der USA 
• Palo Alto, Kalifornien: Internet Software Consortium
192.5.5.250: clock.isc.org
Servicebereich: BARRnet, Alternet-West und CIX-West 
• Cambridge, Massachusetts: Open Software Foundation
130.105.4.59: clock.osf.org
Servicebereich: NSFNET- und NEARnet-Bereich 
• Palo Alto, Kalifornien: ViaNet Communications
209.81.9.7: clock.via.net 
• Cleveland, Ohio: Lewis Research Center (NASA)
128.156.1.43: lerc-dns.lerc.nasa.gov
Servicebereich: NSFNET und OARNET 
• Colorado Springs, Colorado: Schriever AFB
204.34.198.40: navobs1.usnogps.navy.mil; CNAME: tick.usnogps.navy.mil 
204.34.198.41: navobs1.usnogps.navy.mil; CNAME: tock.usnogps.navy.mil 
Servicebereich: US-Zeitzonen PST (Pacific Standard Time) und MST (Mountain Standard Time) 
• St. Louis, Missouri: Washington University
128.252.19.1: navobs1.usnogps.navy.mil; CNAME: tick.wustl.edu 
Servicebereich: US-Zeitzone CST (Central Standard Time) 
• Research Triangle Park, North Carolina: MCNC
192.101.21.1: ncnoc.ncren.net
Servicebereich: NC-REN-Bereich (North Carolina Research and Education Network) 
• Cupertino, Kalifornien: HP
192.6.38.127: ntp-cup.external.hp.com
Servicebereich: USA Westküste 
• Newark, Delaware: Conectiv Communications
138.39.7.20: ntp1.delmarva.com
Servicebereich: Cable & Wireless Network (früher MCInet) 
• University Park, Pennsylvania: Penn State University
128.118.46.3: otc1.psu.edu
Servicebereich: NSFNET, PREPNET und JvNCnet  

Europa
• Borowiec, Polen: Astrogeodynamical Observatory, Space Research Centre
150.254.183.15: vega.cbk.poznan.pl
Servicebereich: Polen und Europa 
• Stockholm, Schweden: Stupi AB
192.36.143.151: Time2.Stupi.SE
Servicebereich: Europa 
• Turin, Italien: IEN Galileo Ferraris
193.204.114.1: time.ien.it
Servicebereich: Italien und Europa 
• Zürich, Schweiz: Integrated Systems Laboratory , Eidgenössischen Technischen Hochschule Zürich 
129.132.2.21: swisstime.ethz.ch
Servicebereich: Schweiz und Europa 
• Turin, Italien: CSTV of National Research Council
150.145.33.1: tempo.cstv.to.cnr.it
Servicebereich: Italien und Europa 
• Erlangen, Deutschland: Universität Erlangen-Nürnberg
ntp0.fau.de; ntp1.fau.de; ntp2.fau.de; 
ntps1-0.uni-erlangen.de; ntps1-1.uni-erlangen.de; ntps1-2.uni-erlangen.de
Servicebereich: Deutschland und Europa 
• Berlin, Deutschland: Technische Universität Berlin
130.149.17.21: ntps1-0.cs.tu-berlin.de
130.149.17.8: ntps1-1.cs.tu-berlin.de
Servicebereich: Deutschland und Europa 
• Deutschland
131.173.17.7: ntps1-1.rz.Uni-Osnabrueck.DE
Servicebereich: Deutschland und Europa 
• Schweden
192.36.143.150: Time1.Stupi.SE
Servicebereich: SUnet und NORDUnet Schweden 

Fernost und pazifische Randgebiete
• Hong Kong: Chinesische Universität von Hong Kong. 
137.189.6.18: clock.cuhk.edu.hk
Servicebereich: Hong Kong (China) und Südostasien  
• Fukuoka, Japan: Universität Fukuoka
133.100.9.2: clock.nc.fukuoka-u.ac.jp
133.100.11.8: clock.tl.fukuoka-u.ac.jp
Servicebereich: Japan und pazifischer Raum  

Australien
• Melbourne, Australien: University of Melbourne
128.250.36.2: ntp.cs.mu.OZ.AU
Servicebereich: Australien und Neuseeland  

Zeitserver der zweiten Ebene
Nach geographischem Standort sortiert: 
Nordamerika
NTP-Zeitserver: • Quebec, Kanada: Canadian Meteorological Center
ntp1.cmc.ec.gc.ca; ntp2.cmc.ec.gc.ca 
Servicebereich: Ostkanada  
• Ontario, Kanada: National Research Council of Canada
time.chu.nrc.ca; time.nrc.ca
Servicebereich: Kanada 
• Saskatchewan, Kanada: University of Regina 
142.3.100.15: timelord.uregina.ca
Servicebereich: Kanada 
• Ontario, Kanada: University of Toronto
tick.utoronto.ca; tock.utoronto.ca
Servicebereich: Ostkanada  
• Mexiko: Audiotel-Büro 
ntp2a.audiotel.com.mx; ntp2c.audiotel.com.mx; ntp2b.audiotel.com.mx
Servicebereich: Avantel, MCINet und Mexiko 
• Santa Cruz, Kalifornien: Scruz-net, inc.
165.227.1.1: ns.scruz.net
Servicebereich: Westen der USA 
• San Diego, Kalifornien: UCSD Academic Computing Services/Network Operations
132.239.254.49: ntp.ucsd.edu
Servicebereich: CERFNET; NSFNET, SDSC-Bereich, und nahegelegene Bereiche 
• Quincy, Kalifornien 
ntp1.mainecoon.com; ntp2.mainecoon.com 
Servicebereich: Nordamerika 
• Newark, Delaware: University of Delaware
128.175.1.3: louie.udel.edu
Servicebereich: CAIRN, Abilene und vBNS  
• Atlanta, Georgia: CNSG
ntp.shorty.com
Servicebereich: Südwesten der USA  
• Kennesaw, Georgia: PeachNet 
rolex.peachnet.edu; timex.peachnet.edu
Servicebereich: PeachNet (Georgia) und Südwesten der USA  
• Urbana-Champaign, Illinois: University of Illinois
ntp-0.cso.uiuc.edu; ntp-1.cso.uiuc.edu; ntp-2.cso.uiuc.edu
Servicebereich: CICNET, Mittlerer Westen und NCSA-Bereich  
• Chicago, Illinois: Argonne National Laboratory 
ntp-1.mcs.anl.gov; ntp-2.mcs.anl.gov
Servicebereich: NSF/ANSNet, CICNet, NetIllinois und ESNet  
• West Lafayette, Indiana: Purdue University
gilbreth.ecn.purdue.edu; harbor.ecn.purdue.edu; molecule.ecn.purdue.edu 
Servicebereich: NSFNET- und CICNET-Bereich  
• Manhattan, Kansas: KansasNet OnLine Services
199.240.130.1: ntp1.kansas.net
199.240.130.12: ntp2.kansas.net
Servicebereich: Zentral-USA und Great Plains  
• Boston, Massachusetts: UMass-Boston CS dept.
158.121.104.4: timeserver.cs.umb.edu
Servicebereich: Neuengland  
• Minneapolis/St Paul, Minnesota: University of Minnesota
ns.nts.umn.edu; nss.nts.umn.edu
Servicebereich: CICNET-Bereich  
• Columbia, Missouri: University of Missouri-Columbia
128.206.206.12: everest.cclabs.missouri.edu
Servicebereich: MOREnet  
• Omaha, Nebraska: Radiks Internet Access
205.138.126.83: allison.radiks.net
Servicebereich: Mittlerer Westen, USA  
• Las Vegas, Nevada: University of Nevada System Computing Services
131.216.1.101: cuckoo.nevada.edu 
Servicebereich: NevadaNet, NSFNET und SDSC-Bereich  
• Las Vegas, Nevada: UNLV College of Engineering
tick.cs.unlv.edu; tock.cs.unlv.edu
Servicebereich: Sprintnet  
• New York City, New York: Columbia University
ntp.ctr.columbia.edu 
Servicebereich: Sprintlink und NYSERnet  
• Ithaca, New York: Cornell University 
192.35.82.50: ntp0.cornell.edu
Servicebereich: NSFNET und NYSER-Bereich  
• New York, New York: Morningside Campus, Columbia University
sundial.columbia.edu
Servicebereich: NYSERnet  
• New York City, New York: Columbia University Computer Science Department
timex.cs.columbia.edu 
Servicebereich: PSINET; NSFNET, und NYSER-Bereich  
• Norman, Oklahoma: University of Oklahoma
129.15.22.8: constellation.ecn.uoknor.edu 
Servicebereich: Midnet  
• Coos Bay, Oregon: Koala Computers
207.48.109.6: tick.koalas.com
Servicebereich: Nordwesten der USA  
• University Park, Pennsylvania: Penn State University
128.118.25.3: clock.psu.edu
Servicebereich: Internet2, vBNS, CERFnet(AT&T IP Services), PSC/NCNE und CASC 
• Pittsburgh, Pennsylvania: Pittsburgh Supercomputing Center
128.182.58.100: fuzz.psc.edu
Servicebereich: NSFNET und PSC-Bereich  
• Pittsburgh, Pennsylvania: Carnegie Mellon Electrical and Computer Engineering 
ntp-1.ece.cmu.edu; ntp-2.ece.cmu.edu 
Servicebereich: PREPNET und PSC-Bereich  
• Dallas, Texas: Cox School of Business, Southern Methodist University
129.119.80.126: ntp.cox.smu.edu 
Servicebereich: NSFNET und SESQUI-Bereich  
• Hughes Springs, Texas: First National Bank
209.144.20.76: ntp.fnbhs.com
Servicebereich: Nordosten Texas  
• Houston, Texas: Baylor College of Medicine
128.249.1.10: ntp.tmc.edu 
Servicebereich: NSFNET und SESQUI-Bereich  
• College Station, Texas: Texas A&M University
165.91.52.110: ntp5.tamu.edu
Servicebereich: NSFNET, SESQUI-Bereich, THEnet und TAMUSDSN 
• Plano, Texas: Greyware Automation Products
tick.greyware.com; tock.greyware.com
Servicebereich: Südzentral-USA  
• Blacksburg, Virginia: Virginia Tech Computing Center
ntp-1.vt.edu; ntp-2.vt.edu
Servicebereich: Südwesten der USA  
• Arlington, Virginia: Center for Seismic Studies
140.162.1.3: ntp.cmr.gov
Servicebereich: NSFNET und SURA-Bereich  
• Richland, Washington: Washington State University 
192.31.216.30: clock.tricity.wsu.edu
Servicebereich: NSFNET und NorthWestNet  
• Washington, USA: Mill Creek
time.ultimeth.net
Servicebereich: Nordwesten der USA  
• Wisconsin, USA: Computer Science Department, University of Wisconsin-Madison
ntp1.cs.wisc.edu; ntp2.cs.wisc.edu; ntp3.cs.wisc.edu
Servicebereich: USA und jeder andere  

Südamerika
• Buenos Aires, Argentinien: Network Access Point
200.49.40.1: CNAME: tick.nap.com.ar
200.49.32.1: CNAME: tock.nap.com.ar
Servicebereich: Argentinien 
• Buenos Aires, Argentinien: Sinectis S.A.
time.sinectis.com.ar 
Servicebereich: Argentinien 
• Brasilien: Brazilian Research Network
200.144.121.33: ntp.cais.rnp.br 
Servicebereich: Brasilien 
• Venezuela: VELUG, Grupo de Usuarios Linux de Venezuela
150.185.192.250: ntp.linux.org.ve
Servicebereich: Arica  

Europa
• Zürich, Schweiz: Eidgenössischen Technischen Hochschule Zürich
129.132.98.11: bernina.ethz.ch
Servicebereich: Schweiz und Europa  
• Standort: Kopenhagen, Dänemark, Europa 
clock.netcetera.dk; clock2.netcetera.dk 
Servicebereich: Dänemark, Skandinavien und Nordeuropa  
• Spanien: Altea 
slug.ctv.es
Servicebereich: Spanien  
• Pieksamaki, Finnland: Keski-Savon Oppimiskeskus
tick.keso.fi; tock.keso.fi
Servicebereich: Finnland  
• Meudon, Frankreich: Observatoire de Paris-Meudon 
ntp.obspm.fr 
Servicebereich: Frankreich und Europa  
• Lyon, Frankreich: CISM 
ntp.univ-lyon1.fr 
Servicebereich: Frankreich, Schweiz, Italien und Europa  
• Paris, Frankreich: VIA, Ecole Centrale
138.195.130.70: ntp.via.ecp.fr
Servicebereich: Frankreich und Europa  
• Budapest, Ungarn: KFKI Research Institute for Particle and Nuclear Physics
148.6.0.1: time.kfki.hu
Servicebereich: HUNGARNET  
• Italien: Net4u Srl, Vercelli, Italien
195.32.52.129: ntps.net4u.it
Servicebereich: Italien  
• Oslo, Norwegen: Universität Oslo
129.240.64.3: fartein.ifi.uio.no 
Servicebereich: NORDUnet  
• Oslo, Norwegen: Alcanet International
time.alcanet.no
Servicebereich: Europa 
• Krakau, Polen: Academic Computer Centre 
149.156.4.11: info.cyf-kr.edu.pl
Servicebereich: Polen und Europa  
• Lund, Schweden: Lund Institute of Technology
130.235.20.3: ntp.lth.se 
Servicebereich: Schweden und NORDUnet 
• Ljubljana, Slowenien: Institute of Biophysics, University of Ljubljana
biofiz.mf.uni-lj.si 193.2.69.11
Servicebereich: Slowenien und Europa  
• Ljubljana, Slowenien: Hydrometeorological Institute of Slovenia
hmljhp.rzs-hm.si
Servicebereich: Slowenien und Europa  
• Ljubljana, Slowenien: Academic and Research Network of Slovenia
ntp1.arnes.si; ntp2.arnes.si
Servicebereich: Slowenien und Europa  
• Ljubljana, Slowenien: J. Stefan Institute
time.ijs.si
Servicebereich: Slowenien und Europa  

Britische Inseln
• Dublin, Irland: School of Mathematics, Trinity College 
ntp.cs.tcd.ie; ntp.maths.tcd.ie; ntp.tcd.ie
Servicebereich: Irland und Großbritannien 
• Glasgow, Schottland: Strathclyde University 
ntp.cs.strath.ac.uk 
Servicebereich: Großbritannien, Europa und andere 
• Cambridge, Großbritannien
ntp0.uk.uu.net; ntp1.uk.uu.net; 
ntp2.uk.uu.net 
Servicebereich: UUNET (in Großbritannien früher auch als PIPEX bekannt) und Großbritannien.  
• Manchester, England: University of Manchester
ntp2a.mcc.ac.uk; ntp2b.mcc.ac.uk;
ntp2c.mcc.ac.uk; ntp2d.mcc.ac.uk 
Servicebereich: Großbritannien  
• Buckinghamshire, Großbritannien: Wibble U.K., Aylesbury
tick.tanac.net
Servicebereich: Großbritannien  

Asien
• Moskau, Russland: Landau Institute for Theoretical Physics
193.233.9.7: ntp.landau.ac.ru
Servicebereich: Russland  
• Russland: Pushchino (bei Moskau)
194.149.67.130: ntp.psn.ru
Servicebereich: Russland 
• Chernogolovka, Russland: Chernogolovka Scientific Center (bei Moskau)
193.233.46.10: sign.chg.ru
Servicebereich: Russland  

Fernost und pazifische Randgebiete
• Tokyo, Japan: Cyber Fleet, Inc.
203.139.30.195: ntp.cyber-fleet.net
Servicebereich: Japan und Ostasien  
• Seoul, Korea: Inet, Inc.
time.nuri.net
Servicebereich: Korea, Japan, Hong Kong und Ostasien  
• Hamilton, Neuseeland: Universität Waikato
truechimer.waikato.ac.nz; truechimer1.waikato.ac.nz; 
truechimer2.waikato.ac.nz; truechimer3.waikato.ac.nz
Servicebereich: Neuseeland  
• Singapur und Philippinen: 
ntp.shim.org 
Servicebereich: Singapur  

Afrika
• Lagos, Nigeria: Supernet300
ntp.supernet300.com
Servicebereich: Westafrika (hauptsächlich nigerischer NITEL-Backbone)  
• Pietermaritzburg, Südafrika: Natal University
143.128.82.200: ntp.cs.unp.ac.za
Servicebereich: Südafrika  

Australien
• Adelaide, Südaustralien: University of Adelaide
129.127.28.4: augean.eleceng.adelaide.edu.au
129.127.40.3: ntp.adelaide.edu.au
203.21.37.18: ntp.saard.net
Servicebereich: AARNet  
• Carlton, Victoria, Australien: eSec Limited
203.21.84.4: time.esec.com.au  

*)

*)
END_FUNCTION_BLOCK

(* POU XTEST/Testprojekt/string_test, ST *)
FUNCTION_BLOCK string_test
VAR_INPUT
END_VAR
VAR_OUTPUT
	good : BOOL;
END_VAR
VAR CONSTANT
	byte1 : BYTE := 1;
END_VAR
VAR
	i: BYTE;
	temp: STRING;
	t: INT;
END_VAR
good := TRUE;

(* test find_char *)
good := good AND FIND_CHAR('1234567890',1) = 1;
good := good AND FIND_CHAR('$03$01gf$023q8t7gq38hg3qzo8gzqo4z7goq8ztgoq3t',3) = 3;
good := good AND FIND_CHAR('$03$01gf$023q8t7gq38hg3qzo8gzqo4z7goq8ztgoq3t',99) = 0;
good := good AND FIND_CHAR('$03$01gf$023q8t7gq38hg3qzo8gzqo4z7goq8ztgoq3t',1) = 3;


(* test is_alnum *)
good := good AND IS_ALNUM('256.188.3.4') = FALSE;
good := good AND IS_ALNUM('02561883479') = TRUE;
good := good AND IS_ALNUM('ABCDEFGHIJKLMNOPQRSTUVWXYZabcdefghijklmnopqrstuvwxyz') = TRUE;
good := good AND IS_ALNUM('sergrsdt[') = FALSE;
good := good AND IS_ALNUM(CHR(47)) = FALSE;
good := good AND IS_ALNUM(CHR(58)) = FALSE;
good := good AND IS_ALNUM(CHR(64)) = FALSE;
good := good AND IS_ALNUM(CHR(91)) = FALSE;
good := good AND IS_ALNUM(CHR(96)) = FALSE;
good := good AND IS_ALNUM(CHR(123)) = FALSE;
good := good AND IS_ALNUM('') = FALSE;


(* test is_alpha *)
good := good AND IS_ALPHA('256.188.3.4') = FALSE;
good := good AND IS_ALPHA('02561883479') = FALSE;
good := good AND IS_ALPHA('ABCDEFGHIJKLMNOPQRSTUVWXYZabcdefghijklmnopqrstuvwxyz') = TRUE;
good := good AND IS_ALPHA('sergrsdt[') = FALSE;
good := good AND IS_ALPHA(CHR(47)) = FALSE;
good := good AND IS_ALPHA(CHR(58)) = FALSE;
good := good AND IS_ALPHA(CHR(64)) = FALSE;
good := good AND IS_ALPHA(CHR(91)) = FALSE;
good := good AND IS_ALPHA(CHR(96)) = FALSE;
good := good AND IS_ALPHA(CHR(123)) = FALSE;
good := good AND IS_ALPHA('') = FALSE;

(* test is_ctrl *)
good := good AND IS_CTRL(CHR(31)) = TRUE;
good := good AND IS_CTRL(CHR(32)) = FALSE;
good := good AND IS_CTRL('') = FALSE;

(* test is_hex *)
good := good AND IS_HEX('abcdef0123456789ABCDEF') = TRUE;
good := good AND IS_HEX('4g') = FALSE;
good := good AND IS_HEX('4G') = FALSE;
good := good AND IS_HEX(CHR(96)) = FALSE;
good := good AND IS_HEX(CHR(64)) = FALSE;
good := good AND IS_HEX(CHR(47)) = FALSE;
good := good AND IS_HEX('') = FALSE;

(* test is_lower *)
good := good AND IS_LOWER('abcdefghijklmnopqrstuvwxyz') = TRUE;
good := good AND IS_LOWER('Dabcdefghijklmnopqrstuvwxyz') = FALSE;
good := good AND IS_LOWER('1abcdefghijklmnopqrstuvwxyz') = FALSE;
good := good AND IS_LOWER('~abcdefghijklmnopqrstuvwxyz') = FALSE;
good := good AND IS_LOWER('') = FALSE;

(* test is_upper *)
good := good AND IS_UPPER('1~ABCDEFGHUIJKLMNOPQRSTUVWXYZ') = FALSE;
good := good AND IS_UPPER('ABCDEFGHUIJKLMNOPQRSTUVWXYZ') = TRUE;
good := good AND IS_UPPER('sABCDEFGHUIJKLMNOPQRSTUVWXYZ') = FALSE;
good := good AND IS_UPPER('') = FALSE;

(* test is_num *)
good := good AND IS_NUM('0123456789') = TRUE;
good := good AND IS_NUM('-0123456789') = FALSE;
good := good AND IS_NUM('a0123456789') = FALSE;
good := good AND IS_NUM('0123456789,') = FALSE;
good := good AND IS_NUM('') = FALSE;

(* test replace_uml *)
good := good AND REPLACE_UML('schußhütte') = 'schusshuette';
good := good AND REPLACE_UML('ÄÖÜäöüß') = 'AeOeUeaeoeuess';
good := good AND REPLACE_UML('blabla') = 'blabla';

(* test byte_to_strb *)
good := good AND BYTE_TO_STRB(INT_TO_BYTE(0)) = '00000000';
good := good AND BYTE_TO_STRB(byte1) = '00000001';
good := good AND BYTE_TO_STRB(SHL(byte1,1)) = '00000010';
good := good AND BYTE_TO_STRB(SHL(byte1,2)) = '00000100';
good := good AND BYTE_TO_STRB(SHL(byte1,3)) = '00001000';
good := good AND BYTE_TO_STRB(SHL(byte1,4)) = '00010000';
good := good AND BYTE_TO_STRB(SHL(byte1,5)) = '00100000';
good := good AND BYTE_TO_STRB(SHL(byte1,6)) = '01000000';
good := good AND BYTE_TO_STRB(SHL(byte1,7)) = '10000000';
good := good AND BYTE_TO_STRB(INT_TO_BYTE(255)) = '11111111';

(* test byte_to_strh *)
good := good AND BYTE_TO_STRH(INT_TO_BYTE(0)) = '00';
good := good AND BYTE_TO_STRH(byte1) = '01';
good := good AND BYTE_TO_STRH(SHL(byte1,1)) = '02';
good := good AND BYTE_TO_STRH(SHL(byte1,2)) = '04';
good := good AND BYTE_TO_STRH(SHL(byte1,3)) = '08';
good := good AND BYTE_TO_STRH(SHL(byte1,4)) = '10';
good := good AND BYTE_TO_STRH(SHL(byte1,5)) = '20';
good := good AND BYTE_TO_STRH(SHL(byte1,6)) = '40';
good := good AND BYTE_TO_STRH(SHL(byte1,7)) = '80';
good := good AND BYTE_TO_STRH(INT_TO_BYTE(255)) = 'FF';

(* test chr function *)
good := good AND CHR(32) = ' ';
good := good AND CHR(44) = ',';
good := good AND CHR(54) = '6';
good := good AND CHR(74) = 'J';
good := good AND CHR(104) = 'h';

(* test dword_to_strb *)
good := good AND DWORD_TO_STRB(0) = '00000000000000000000000000000000';
good := good AND DWORD_TO_STRB(256) = '00000000000000000000000100000000';


(* test dword_to_strh *)
good := good AND DWORD_TO_STRH(0) = '00000000';
good := good AND DWORD_TO_STRH(256) = '00000100';

(* test dword_to_strf *)
good := good AND DWORD_TO_STRF(0,3) = '000';
good := good AND DWORD_TO_STRF(4567,3) = '567';
good := good AND DWORD_TO_STRF(3,3) = '003';
good := good AND DWORD_TO_STRF(0,0) = '';

(* test exec *)
good := good AND EXEC('2/0') = 'ERROR';
good := good AND EXEC('2/2') = '1.0';
good := good AND EXEC('2+2') = '4.0';
good := good AND EXEC('2-2') = '0.0';
good := good AND EXEC('2*2') = '4.0';
good := good AND EXEC('2^2') = '4.0';
good := good AND EXEC('SQRT4') = '2.0';

(* test count_char *)
good := good AND COUNT_CHAR(' sdfg wse   rgt ert',32) = 6;

(* test find_ctrl *)
good := good AND FIND_CTRL('1234$0A567890',1) = 5;
good := good AND FIND_CTRL('1234$0A567890',5) = 5;
good := good AND FIND_CTRL('1234$0A567890',6) = 0;
good := good AND FIND_CTRL('1234567890',1) = 0;


(* test find_nonum *)
good := good AND FIND_NONUM('1234n3643n5',1) = 5;
good := good AND FIND_NONUM('1234n3643n5',5) = 5;
good := good AND FIND_NONUM('1234n3643n5',6) = 10;
good := good AND FIND_NONUM('123436435',1) = 0;

(* test find_num *)
good := good AND FIND_NUM('abc4eg',1) = 4;
good := good AND FIND_NUM('abc4eg',4) = 4;
good := good AND FIND_NUM('abc4eg',5) = 0;
good := good AND FIND_NUM('abceg',1) = 0;

(* test findB *)
good := good AND FINDB('abcdabcd','ab') = 5;
good := good AND FINDB('abcdabcd','ba') = 0;

(* test FINDB_NONUM *)
good := good AND FINDB_NONUM('d2d3456') = 3;
good := good AND FINDB_NONUM('23456') = 0;

(* test FINDB_NUM *)
good := good AND FINDB_NUM('2abcd2ef') = 6;
good := good AND FINDB_NUM('absdrfger') = 0;

(* test findp *)
good := good AND FINDP('abcdeabcde','bc',2) = 2;
good := good AND FINDP('abcdeabcde','bc',3) = 7;
good := good AND FINDP('abcdeabcde','bc',7) = 7;
good := good AND FINDP('abcdeabcde','bc',8) = 0;

(* test hex_to_dword *)
good := good AND HEX_TO_DWORD('0ff') = 255;
good := good AND HEX_TO_DWORD('00') = 0;
good := good AND HEX_TO_DWORD('1') = 1;
good := good AND HEX_TO_DWORD('0A') = 10;
good := good AND HEX_TO_DWORD('0F') = 15;
good := good AND HEX_TO_DWORD('0a') = 10;
good := good AND HEX_TO_DWORD('0f') = 15;
good := good AND HEX_TO_DWORD('00009') = 9;

(* test lowercase *)
good := good AND LOWERCASE('FGTHZuz2345KJGH') = 'fgthzuz2345kjgh';

(* test mirror *)
good := good AND MIRROR('123456789 abc') = 'cba 987654321';

(* test real_to_strf *)
good := good AND REAL_TO_STRF(pi1,2) = '3.14';
good := good AND REAL_TO_STRF(0.015,2) = '0.02';
good := good AND REAL_TO_STRF(0.015,4) = '0.0150';
good := good AND REAL_TO_STRF(0.015,0) = '0';
good := good AND REAL_TO_STRF(3.015,1) = '3.0';
good := good AND REAL_TO_STRF(1234.49967,0) = '1234';
good := good AND REAL_TO_STRF(1234.49967,1) = '1234.5';
good := good AND REAL_TO_STRF(1234.49967,2) = '1234.50';
good := good AND REAL_TO_STRF(1234.49964,3) = '1234.500';
good := good AND REAL_TO_STRF(14.49967,4) = '14.4997';
good := good AND REAL_TO_STRF(1.49967,5) = '1.49967';
good := good AND REAL_TO_STRF(1.49967,6) = '1.499670';

(* test replace_all *)
good := good AND REPLACE_ALL('ab12cd12ef12gh','12','') = 'abcdefgh';
good := good AND REPLACE_ALL('ab12cd12ef12gh','12','21') = 'ab21cd21ef21gh';
good := good AND REPLACE_ALL('ab12cd12ef12gh','12','12') = 'ab12cd12ef12gh';

(* test trim *)
good := good AND TRIM(' ab  cd ef  gh ') = 'abcdefgh';


(* test trim1 *)
good := good AND TRIM1(' ab  cd ef  gh ') = 'ab cd ef gh';

(* test uppercase *)
good := good AND UPPERCASE('fgTHZu z2345KJGH') = 'FGTHZU Z2345KJGH';

(* test capitalize *)
good := good AND CAPITALIZE('hugo wallenstein 123') = 'Hugo Wallenstein 123';

(* test to_upper and to lower *)
FOR t := 0 TO 255 DO
	i := INT_TO_BYTE(t);
	CASE i OF
	0..64:
		good := good AND TO_LOWER(i) = i AND TO_UPPER(i) = i;
	65..90: (* uppercase letters *)
		good := good AND TO_UPPER(i) = i;
		good := good AND TO_LOWER(i) = i + 32;
	91..96:
		good := good AND TO_LOWER(i) = i AND TO_UPPER(i) = i;
	97..122: (* small letters *)
		good := good AND TO_UPPER(i) = i - 32;
		good := good AND TO_LOWER(i) = i;
	123..191:
		good := good AND TO_LOWER(i) = i AND TO_UPPER(i) = i;
	192..214: (* extended uppercase letters *)
		good := good AND TO_UPPER(i) = i;
		good := good AND TO_LOWER(i) = i + 32;
	215:
		good := good AND TO_LOWER(i) = i AND TO_UPPER(i) = i;
	216..222: (* extended uppercase letters *)
		good := good AND TO_UPPER(i) = i;
		good := good AND TO_LOWER(i) = i + 32;
	223:
		good := good AND TO_LOWER(i) = i AND TO_UPPER(i) = i;
	224..246: (* extended lowercase letters *)
		good := good AND TO_UPPER(i) = i-32;
		good := good AND TO_LOWER(i) = i;
	247:
		good := good AND TO_LOWER(i) = i AND TO_UPPER(i) = i;
	248..254: (* extended lowercase letters *)
		good := good AND TO_UPPER(i) = i-32;
		good := good AND TO_LOWER(i) = i;
	255:
		good := good AND TO_LOWER(i) = i AND TO_UPPER(i) = i;
	END_CASE;
	temp := CONCAT(INT_TO_STRING(t),' > ');
	temp := CONCAT(temp,CHR(TO_UPPER(i)));
	temp := CONCAT(temp,' > ');
	temp := CONCAT(temp,CHR(TO_LOWER(i)));
END_FOR;

(* test isc funktionen *)
FOR t := 0 TO 255 DO
	i := INT_TO_BYTE(t);
	CASE i OF
	0..31:
		good := good AND ISC_CTRL(i) = TRUE;
		good := good AND ISC_NUM(i) = FALSE;
		good := good AND ISC_ALPHA(i) = FALSE;
		good := good AND ISC_HEX(i) = FALSE;
		good := good AND ISC_LOWER(i) = FALSE;
		good := good AND ISC_UPPER(i) = FALSE;
	32..47:
		good := good AND ISC_CTRL(i) = FALSE;
		good := good AND ISC_NUM(i) = FALSE;
		good := good AND ISC_ALPHA(i) = FALSE;
		good := good AND ISC_HEX(i) = FALSE;
		good := good AND ISC_LOWER(i) = FALSE;
		good := good AND ISC_UPPER(i) = FALSE;
	48..57:
		good := good AND ISC_CTRL(i) = FALSE;
		good := good AND ISC_NUM(i) = TRUE;
		good := good AND ISC_ALPHA(i) = FALSE;
		good := good AND ISC_HEX(i) = TRUE;
		good := good AND ISC_LOWER(i) = FALSE;
		good := good AND ISC_UPPER(i) = FALSE;
	58..64:
		good := good AND ISC_CTRL(i) = FALSE;
		good := good AND ISC_NUM(i) = FALSE;
		good := good AND ISC_ALPHA(i) = FALSE;
		good := good AND ISC_HEX(i) = FALSE;
		good := good AND ISC_LOWER(i) = FALSE;
		good := good AND ISC_UPPER(i) = FALSE;
	65..70:
		good := good AND ISC_CTRL(i) = FALSE;
		good := good AND ISC_NUM(i) = FALSE;
		good := good AND ISC_ALPHA(i) = TRUE;
		good := good AND ISC_HEX(i) = TRUE;
		good := good AND ISC_LOWER(i) = FALSE;
		good := good AND ISC_UPPER(i) = TRUE;
	75..90:
		good := good AND ISC_CTRL(i) = FALSE;
		good := good AND ISC_NUM(i) = FALSE;
		good := good AND ISC_ALPHA(i) = TRUE;
		good := good AND ISC_HEX(i) = FALSE;
		good := good AND ISC_LOWER(i) = FALSE;
		good := good AND ISC_UPPER(i) = TRUE;
	91..96:
		good := good AND ISC_CTRL(i) = FALSE;
		good := good AND ISC_NUM(i) = FALSE;
		good := good AND ISC_ALPHA(i) = FALSE;
		good := good AND ISC_HEX(i) = FALSE;
		good := good AND ISC_LOWER(i) = FALSE;
		good := good AND ISC_UPPER(i) = FALSE;
	97..102:
		good := good AND ISC_CTRL(i) = FALSE;
		good := good AND ISC_NUM(i) = FALSE;
		good := good AND ISC_ALPHA(i) = TRUE;
		good := good AND ISC_HEX(i) = TRUE;
		good := good AND ISC_LOWER(i) = TRUE;
		good := good AND ISC_UPPER(i) = FALSE;
	103..122:
		good := good AND ISC_CTRL(i) = FALSE;
		good := good AND ISC_NUM(i) = FALSE;
		good := good AND ISC_ALPHA(i) = TRUE;
		good := good AND ISC_HEX(i) = FALSE;
		good := good AND ISC_LOWER(i) = TRUE;
		good := good AND ISC_UPPER(i) = FALSE;
	123..126:
		good := good AND ISC_CTRL(i) = FALSE;
		good := good AND ISC_NUM(i) = FALSE;
		good := good AND ISC_ALPHA(i) = FALSE;
		good := good AND ISC_HEX(i) = FALSE;
		good := good AND ISC_LOWER(i) = FALSE;
		good := good AND ISC_UPPER(i) = FALSE;
	127:
		good := good AND ISC_CTRL(i) = TRUE;
		good := good AND ISC_NUM(i) = FALSE;
		good := good AND ISC_ALPHA(i) = FALSE;
		good := good AND ISC_HEX(i) = FALSE;
		good := good AND ISC_LOWER(i) = FALSE;
		good := good AND ISC_UPPER(i) = FALSE;
	128..191:
		good := good AND ISC_CTRL(i) = FALSE;
		good := good AND ISC_NUM(i) = FALSE;
		good := good AND ISC_ALPHA(i) = FALSE;
		good := good AND ISC_HEX(i) = FALSE;
		good := good AND ISC_LOWER(i) = FALSE;
		good := good AND ISC_UPPER(i) = FALSE;
	192..214:
		good := good AND ISC_CTRL(i) = FALSE;
		good := good AND ISC_NUM(i) = FALSE;
		good := good AND ISC_ALPHA(i) = EXTENDED_ASCII;
		good := good AND ISC_HEX(i) = FALSE;
		good := good AND ISC_LOWER(i) = FALSE;
		good := good AND ISC_UPPER(i) = EXTENDED_ASCII;
	215:
		good := good AND ISC_CTRL(i) = FALSE;
		good := good AND ISC_NUM(i) = FALSE;
		good := good AND ISC_ALPHA(i) = FALSE;
		good := good AND ISC_HEX(i) = FALSE;
		good := good AND ISC_LOWER(i) = FALSE;
		good := good AND ISC_UPPER(i) = FALSE;
	216..222:
		good := good AND ISC_CTRL(i) = FALSE;
		good := good AND ISC_NUM(i) = FALSE;
		good := good AND ISC_ALPHA(i) = EXTENDED_ASCII;
		good := good AND ISC_HEX(i) = FALSE;
		good := good AND ISC_LOWER(i) = FALSE;
		good := good AND ISC_UPPER(i) = EXTENDED_ASCII;
	223:
		good := good AND ISC_CTRL(i) = FALSE;
		good := good AND ISC_NUM(i) = FALSE;
		good := good AND ISC_ALPHA(i) = TRUE;
		good := good AND ISC_HEX(i) = FALSE;
		good := good AND ISC_LOWER(i) = TRUE;
		good := good AND ISC_UPPER(i) = FALSE;
	224..246:
		good := good AND ISC_CTRL(i) = FALSE;
		good := good AND ISC_NUM(i) = FALSE;
		good := good AND ISC_ALPHA(i) = EXTENDED_ASCII;
		good := good AND ISC_HEX(i) = FALSE;
		good := good AND ISC_LOWER(i) = EXTENDED_ASCII;
		good := good AND ISC_UPPER(i) = FALSE;
	247:
		good := good AND ISC_CTRL(i) = FALSE;
		good := good AND ISC_NUM(i) = FALSE;
		good := good AND ISC_ALPHA(i) = FALSE;
		good := good AND ISC_HEX(i) = FALSE;
		good := good AND ISC_LOWER(i) = FALSE;
		good := good AND ISC_UPPER(i) = FALSE;
	248..254:
		good := good AND ISC_CTRL(i) = FALSE;
		good := good AND ISC_NUM(i) = FALSE;
		good := good AND ISC_ALPHA(i) = EXTENDED_ASCII;
		good := good AND ISC_HEX(i) = FALSE;
		good := good AND ISC_LOWER(i) = EXTENDED_ASCII;
		good := good AND ISC_UPPER(i) = FALSE;
	255:
		good := good AND ISC_CTRL(i) = FALSE;
		good := good AND ISC_NUM(i) = FALSE;
		good := good AND ISC_ALPHA(i) = TRUE;
		good := good AND ISC_HEX(i) = FALSE;
		good := good AND ISC_LOWER(i) = TRUE;
		good := good AND ISC_UPPER(i) = FALSE;
	END_CASE;
END_FOR;

(* code test *)
FOR t := 1 TO 255 DO
	good := good AND CODE(CHR(INT_TO_BYTE(t)),1) = INT_TO_BYTE(t);
END_FOR;
temp := '0123456789';
good := good AND CODE(temp,1) = 48;
good := good AND CODE(temp,0) = 0;
good := good AND CODE(temp,11) = 0;
good := good AND CODE(temp,10) = 57;
END_FUNCTION_BLOCK

(* POU String/TRIM1, ST *)
FUNCTION TRIM1 : STRING
VAR_INPUT
	str : STRING;
END_VAR
VAR
	pos: INT;
END_VAR

(*
version 1.0	4 feb 2008
programmer 	hugo
tested by		tobias

the function replaces all multiple blanks within a string by only one blank.
leading and ending blanks will be deleted

*)
trim1 := str;
REPEAT
	pos := FIND(trim1,'  ');
	trim1 := REPLACE(trim1,' ',2,pos);
UNTIL pos = 0	END_REPEAT;
(* beginning and ending blanks need to be stripped off *)
IF LEFT(trim1,1) = ' ' THEN trim1 := DELETE(trim1,1,1); END_IF;
IF RIGHT(trim1,1) = ' ' THEN trim1 := DELETE(trim1,1,LEN(trim1)); END_IF;


(* revision histroy
hm		4. feb. 2008		rev 1.0
	original release

*)	
END_FUNCTION

(* POU Logic/gate logic/Swap_Byte, ST *)
FUNCTION Swap_Byte : WORD
VAR_INPUT
	IN : WORD;
END_VAR
VAR
END_VAR

(*
version 1.0	4 feb 2008
programmer 	hugo
tested by		tobias

This function swaps the high and low byte of the word in.

*)
Swap_Byte := ROL(in,8);


(* revision history
hm		4. feb 2008	rev 1.0
	original version

*)
END_FUNCTION

(* POU Logic/gate logic/Swap_Byte2, ST *)
FUNCTION Swap_Byte2 : DWORD
VAR_INPUT
	IN : DWORD;
END_VAR
VAR
END_VAR

(*
version 1.0	4 feb 2008
programmer 	hugo
tested by		tobias

This function reverses the byte order in the dword.

*)
Swap_Byte2 := (ROR(in,8) AND 16#FF00FF00) OR (ROL(in,8) AND 16#00FF00FF);

(* revision history
hm		4. feb 2008	rev 1.0
	original version

*)
END_FUNCTION

(* POU Engineering/measurements/TC_MS, ST *)
FUNCTION_BLOCK TC_MS
VAR_INPUT
END_VAR
VAR_OUTPUT
	TC : DWORD;
END_VAR
VAR
	init: BOOL;
	tx: DWORD;
	last: DWORD;
END_VAR

(*
	version 1.0	13 mar 2008
	programmer 	hugo
	tested by		tobias

TC_MS delivers the time it was last called on the output TC in Milliseconds.

*)
(* read system timer *)
tx := T_PLC_MS();

IF NOT init THEN
	init := TRUE;
	TC := 0;
ELSE
	tc := tx - last;
END_IF;
last := tx;

(* revision history
hm		13. mar. 2008	rev 1.0
	original version

*)
END_FUNCTION_BLOCK

(* POU Engineering/measurements/TC_US, ST *)
FUNCTION_BLOCK TC_US
VAR_INPUT
END_VAR
VAR_OUTPUT
	TC : DWORD;
END_VAR
VAR
	init: BOOL;
	tx: DWORD;
	last: DWORD;
END_VAR

(*
	version 1.0	13 mar 2008
	programmer 	hugo
	tested by		tobias

TC_US delivers the time it was last called on the output TC in Microseconds.

*)
(* read system timer *)
tx := T_PLC_US();

IF NOT init THEN
	init := TRUE;
	TC := 0;
ELSE
	tc := tx - last;
END_IF;
last := tx;

(* revision history
hm		13. mar. 2008	rev 1.0
	original version

*)
END_FUNCTION_BLOCK

(* POU Logic/generators/TONOF, ST *)
FUNCTION_BLOCK TONOF
VAR_INPUT
	IN : BOOL;
	T1, T2 : TIME;
END_VAR
VAR_OUTPUT
	Q : BOOL;
END_VAR
VAR
	X : TON;
	Y : TOF;
END_VAR

(*
version 1.1	17 sep 2007
programmer 	hugo
tested by		tobias

TONOF generated a TON and TOF Delay for the Input N TON (T1) and TOF (T2) can be configured separately
*)
X(IN := IN, PT := T1);
Y(in := X.Q, PT := T2);
Q := Y.Q;

(* revision history
hm	10. dec 2007	rev 1.0
	original version

*)
	
END_FUNCTION_BLOCK

(* POU Engineering/signal processing/Word_to_Range, ST *)
FUNCTION Word_to_Range : REAL
VAR_INPUT
	X : WORD;
	low : REAL;
	high : REAL;
END_VAR
VAR
END_VAR

(*
version 1.0	9. jan 2008
programmer 	hugo
tested by		tobias

Word_to_Range converts a Byte into a real between low and high.

*)
Word_to_Range := (high - low) * X / 65535.0 + low;


(* revision history
hm	9. jan 2008		rev 1.0
	original version

*)
END_FUNCTION

(* POU XTEST/Baustein Tests/work_week_test, ST *)
FUNCTION_BLOCK work_week_test
VAR_INPUT
END_VAR
VAR_OUTPUT
	error : BOOL;
	dx: DATE;
END_VAR
VAR
	y : ARRAY[0..30] OF INT := 1990,1991,1992,1993,1993,1994,1994,1995,1995,1996,1997,1998,1999,1999,2000,2000,2001,2002,2003,2004,2005,2005,2006,2006,2007,2008,2009,2010,2010,2011,2011;
	w : ARRAY[0..30] OF INT := 1,	1,	 1,   53,  1,   52,	 1,   52,  1,   1,   1,   1,   53,  1,   52,  1,   1,   1,   1,   1,   53,  1,   52,  1,   1,	1,   1,	  53,  1,   52,  1;
	d : ARRAY[0..30] OF INT := 7,	6,	 5,	  3,   10,  2,   9,   1,   8,   7,   5,   4,   3,   10,  2,   9,   7,   6,   5,   4,   2,   9,   1,   8,   7,	6,	 4,	  3,   10,  2,   9;
	i: INT;
	comp: INT;
	d1: DATE;
	day: INT;
	week: INT;
	yr: INT;
END_VAR
IF error THEN RETURN; END_IF;

FOR i := 0 TO 30 DO
	day := d[i];
	week := w[i];
	yr := y[i];
	d1 := set_Date(yr,1,day);
	comp := work_week(d1);
	IF comp <> week THEN
		error := TRUE;
		dx := d1;
	END_IF;
	d1 := date_add(d1,-6,0,0,0);
	comp := work_week(d1);
	IF comp <> week THEN
		error := TRUE;
		dx := d1;
	END_IF;

END_FOR;
END_FUNCTION_BLOCK

(* POU XTEST/Baustein Tests/year_test, ST *)
FUNCTION year_test : BOOL
VAR_INPUT
END_VAR
VAR
	x : BOOL := TRUE;
	i: INT;
	jan1: DATE;
	dez31: DATE;
END_VAR
FOR i := 1980 TO 2099 DO
	jan1 := set_Date(i,1,1);
	dez31 := set_Date(i,12,31);
	x := X AND year(jan1) = i AND year(dez31) = i;
END_FOR;
year_test := x;
END_FUNCTION
